LIN {X 0,Y 362.292,Z 979.123,A -85,B 0,C 180,E1 20647.364,E2 20647.364} C_VEL
LIN {X 0,Y 378.489,Z 944.913,A -85,B 0,C 180,E1 20652.896,E2 20652.896} C_VEL
LIN {X 0,Y 394.767,Z 905.956,A -85,B 0,C 180,E1 20657.324,E2 20657.324} C_VEL
LIN {X 0,Y 409.414,Z 863.634,A -85,B 0,C 180,E1 20660.691,E2 20660.691} C_VEL
LIN {X 0,Y 410.209,Z 859.007,A -85,B 0,C 180,E1 20661.092,E2 20661.092} C_VEL
LIN {X 0,Y 403.071,Z 830.26,A -85,B 0,C 180,E1 20665.806,E2 20665.806} C_VEL
LIN {X 0,Y 392.847,Z 803.519,A -85,B 0,C 180,E1 20671.168,E2 20671.168} C_VEL
LIN {X 0,Y 382.357,Z 782.646,A -85,B 0,C 180,E1 20676.647,E2 20676.647} C_VEL
LIN {X 0,Y 373.302,Z 766.723,A -85,B 0,C 180,E1 20682.27,E2 20682.27} C_VEL
LIN {X 0,Y 368.306,Z 759.241,A -85,B 0,C 180,E1 20686.159,E2 20686.159} C_VEL
LIN {X 0,Y 364.911,Z 753.277,A -85,B 0,C 180,E1 20689.83,E2 20689.83} C_VEL
LIN {X 0,Y 361.485,Z 746.529,A -85,B 0,C 180,E1 20698.795,E2 20698.795} C_VEL
LIN {X 0,Y 361.688,Z 747.798,A -85,B 0,C 180,E1 20701.421,E2 20701.421} C_VEL
LIN {X 0,Y 366.173,Z 754.902,A -85,B 0,C 180,E1 20709.074,E2 20709.074} C_VEL
LIN {X 0,Y 371.126,Z 763.095,A -85,B 0,C 180,E1 20713.499,E2 20713.499} C_VEL
LIN {X 0,Y 378.632,Z 774.835,A -85,B 0,C 180,E1 20718.367,E2 20718.367} C_VEL
LIN {X 0,Y 390.26,Z 795.362,A -85,B 0,C 180,E1 20724.362,E2 20724.362} C_VEL
LIN {X 0,Y 401.792,Z 821.282,A -85,B 0,C 180,E1 20729.832,E2 20729.832} C_VEL
LIN {X 0,Y 411.136,Z 849.862,A -85,B 0,C 180,E1 20734.599,E2 20734.599} C_VEL
LIN {X 0,Y 413.088,Z 859.947,A -85,B 0,C 180,E1 20735.992,E2 20735.992} C_VEL
LIN {X 0,Y 398.616,Z 904.569,A -85,B 0,C 180,E1 20738.996,E2 20738.996} C_VEL
LIN {X 0,Y 382.398,Z 945.744,A -85,B 0,C 180,E1 20743.057,E2 20743.057} C_VEL
LIN {X 0,Y 366.082,Z 981.986,A -85,B 0,C 180,E1 20748.161,E2 20748.161} C_VEL
LIN {X 0,Y 351.337,Z 1013.074,A -85,B 0,C 180,E1 20754.389,E2 20754.389} C_VEL
LIN {X 0,Y 339.93,Z 1037.627,A -85,B 0,C 180,E1 20761.363,E2 20761.363} C_VEL
LIN {X 0,Y 332.379,Z 1056.352,A -85,B 0,C 180,E1 20769.02,E2 20769.02} C_VEL
LIN {X 0,Y 328.863,Z 1068.693,A -85,B 0,C 180,E1 20776.678,E2 20776.678} C_VEL
LIN {X 0,Y 328.034,Z 1074.064,A -85,B 0,C 180,E1 20782.033,E2 20782.033} C_VEL
LIN {X 0,Y 328.003,Z 1077.219,A -85,B 0,C 180,E1 20789.999,E2 20789.999} C_VEL
LIN {X 0,Y 327.96,Z 1074.585,A -85,B 0,C 180,E1 20797.967,E2 20797.967} C_VEL
LIN {X 0,Y 329.425,Z 1067.671,A -85,B 0,C 180,E1 20804.999,E2 20804.999} C_VEL
LIN {X 0,Y 334.439,Z 1053.272,A -85,B 0,C 180,E1 20813.357,E2 20813.357} C_VEL
LIN {X 0,Y 344.133,Z 1032.137,A -85,B 0,C 180,E1 20821.314,E2 20821.314} C_VEL
LIN {X 0,Y 357.491,Z 1005.639,A -85,B 0,C 180,E1 20828.176,E2 20828.176} C_VEL
LIN {X 0,Y 372.702,Z 975.355,A -85,B 0,C 180,E1 20833.725,E2 20833.725} C_VEL
LIN {X 0,Y 388.88,Z 940.762,A -85,B 0,C 180,E1 20838.265,E2 20838.265} C_VEL
LIN {X 0,Y 404.573,Z 902.35,A -85,B 0,C 180,E1 20841.866,E2 20841.866} C_VEL
LIN {X 0,Y 418.082,Z 861.927,A -85,B 0,C 180,E1 20844.559,E2 20844.559} C_VEL
LIN {X 0,Y 409.957,Z 833.961,A -85,B 0,C 180,E1 20849.35,E2 20849.35} C_VEL
LIN {X 0,Y 399.624,Z 808.583,A -85,B 0,C 180,E1 20854.842,E2 20854.842} C_VEL
LIN {X 0,Y 393.435,Z 796.515,A -85,B 0,C 180,E1 20858.246,E2 20858.246} C_VEL
LIN {X 0,Y 389.709,Z 795.233,A -85,B 0,C 180,E1 20859.866,E2 20859.866} C_VEL
LIN {X 0,Y 386.052,Z 794.568,A -85,B 0,C 180,E1 20861.545,E2 20861.545} C_VEL
LIN {X 0,Y 378.893,Z 781.987,A -85,B 0,C 180,E1 20867.338,E2 20867.338} C_VEL
LIN {X 0,Y 375.953,Z 776.169,A -85,B 0,C 180,E1 20871.018,E2 20871.018} C_VEL
LIN {X 0,Y 373.294,Z 769.834,A -85,B 0,C 180,E1 20879.423,E2 20879.423} C_VEL
LIN {X 0,Y 376.486,Z 777.904,A -85,B 0,C 180,E1 20888.613,E2 20888.613} C_VEL
LIN {X 0,Y 380.579,Z 785.858,A -85,B 0,C 180,E1 20893.093,E2 20893.093} C_VEL
LIN {X 0,Y 386.293,Z 796.722,A -85,B 0,C 180,E1 20897.704,E2 20897.704} C_VEL
LIN {X 0,Y 394.613,Z 814.838,A -85,B 0,C 180,E1 20903.244,E2 20903.244} C_VEL
LIN {X 0,Y 402.714,Z 837.776,A -85,B 0,C 180,E1 20908.5,E2 20908.5} C_VEL
LIN {X 0,Y 408.935,Z 862.896,A -85,B 0,C 180,E1 20913.197,E2 20913.197} C_VEL
LIN {X 0,Y 408.939,Z 868.346,A -85,B 0,C 180,E1 20913.956,E2 20913.956} C_VEL
LIN {X 0,Y 394.051,Z 907.639,A -85,B 0,C 180,E1 20917.064,E2 20917.064} C_VEL
LIN {X 0,Y 376.826,Z 945.755,A -85,B 0,C 180,E1 20921.379,E2 20921.379} C_VEL
LIN {X 0,Y 359.627,Z 979.236,A -85,B 0,C 180,E1 20926.786,E2 20926.786} C_VEL
LIN {X 0,Y 343.841,Z 1008.047,A -85,B 0,C 180,E1 20933.49,E2 20933.49} C_VEL
LIN {X 0,Y 332.266,Z 1029.329,A -85,B 0,C 180,E1 20940.642,E2 20940.642} C_VEL
LIN {X 0,Y 325.06,Z 1044.409,A -85,B 0,C 180,E1 20948.104,E2 20948.104} C_VEL
LIN {X 0,Y 321.603,Z 1053.264,A -85,B 0,C 180,E1 20954.699,E2 20954.699} C_VEL
LIN {X 0,Y 319.956,Z 1058.652,A -85,B 0,C 180,E1 20961.833,E2 20961.833} C_VEL
LIN {X 0,Y 320.103,Z 1059.662,A -85,B 0,C 180,E1 20970.001,E2 20970.001} C_VEL
LIN {X 0,Y 320.678,Z 1055.234,A -85,B 0,C 180,E1 20978.151,E2 20978.151} C_VEL
LIN {X 0,Y 323.464,Z 1046.348,A -85,B 0,C 180,E1 20985.629,E2 20985.629} C_VEL
LIN {X 0,Y 329.929,Z 1030.99,A -85,B 0,C 180,E1 20993.549,E2 20993.549} C_VEL
LIN {X 0,Y 340.701,Z 1009.055,A -85,B 0,C 180,E1 21001.137,E2 21001.137} C_VEL
LIN {X 0,Y 354.739,Z 981.771,A -85,B 0,C 180,E1 21007.676,E2 21007.676} C_VEL
LIN {X 0,Y 370.156,Z 950.547,A -85,B 0,C 180,E1 21012.981,E2 21012.981} C_VEL
LIN {X 0,Y 385.613,Z 915.656,A -85,B 0,C 180,E1 21017.257,E2 21017.257} C_VEL
LIN {X 0,Y 400.393,Z 876.252,A -85,B 0,C 180,E1 21020.729,E2 21020.729} C_VEL
LIN {X 0,Y 404.623,Z 862.747,A -85,B 0,C 180,E1 21021.704,E2 21021.704} C_VEL
LIN {X 0,Y 397.926,Z 834.187,A -85,B 0,C 180,E1 21026.549,E2 21026.549} C_VEL
LIN {X 0,Y 388.172,Z 807.746,A -85,B 0,C 180,E1 21032.061,E2 21032.061} C_VEL
LIN {X 0,Y 377.812,Z 785.992,A -85,B 0,C 180,E1 21038.078,E2 21038.078} C_VEL
LIN {X 0,Y 369.588,Z 772.075,A -85,B 0,C 180,E1 21043.714,E2 21043.714} C_VEL
LIN {X 0,Y 366.487,Z 766.793,A -85,B 0,C 180,E1 21046.394,E2 21046.394} C_VEL
LIN {X 0,Y 363.309,Z 760.907,A -85,B 0,C 180,E1 21050.088,E2 21050.088} C_VEL
LIN {X 0,Y 360.349,Z 754.316,A -85,B 0,C 180,E1 21058.791,E2 21058.791} C_VEL
LIN {X 0,Y 360.53,Z 755.742,A -85,B 0,C 180,E1 21061.426,E2 21061.426} C_VEL
LIN {X 0,Y 364.652,Z 762.65,A -85,B 0,C 180,E1 21068.886,E2 21068.886} C_VEL
LIN {X 0,Y 369.221,Z 770.705,A -85,B 0,C 180,E1 21073.268,E2 21073.268} C_VEL
LIN {X 0,Y 376.265,Z 782.283,A -85,B 0,C 180,E1 21078.107,E2 21078.107} C_VEL
LIN {X 0,Y 386.877,Z 802.016,A -85,B 0,C 180,E1 21083.973,E2 21083.973} C_VEL
LIN {X 0,Y 397.578,Z 827.186,A -85,B 0,C 180,E1 21089.384,E2 21089.384} C_VEL
LIN {X 0,Y 405.873,Z 854.347,A -85,B 0,C 180,E1 21094.054,E2 21094.054} C_VEL
LIN {X 0,Y 407.499,Z 862.634,A -85,B 0,C 180,E1 21095.268,E2 21095.268} C_VEL
LIN {X 0,Y 393.211,Z 905.194,A -85,B 0,C 180,E1 21098.169,E2 21098.169} C_VEL
LIN {X 0,Y 376.403,Z 946.465,A -85,B 0,C 180,E1 21102.286,E2 21102.286} C_VEL
LIN {X 0,Y 359.289,Z 983.156,A -85,B 0,C 180,E1 21107.557,E2 21107.557} C_VEL
LIN {X 0,Y 344.063,Z 1014.027,A -85,B 0,C 180,E1 21113.906,E2 21113.906} C_VEL
LIN {X 0,Y 331.885,Z 1039.267,A -85,B 0,C 180,E1 21121.35,E2 21121.35} C_VEL
LIN {X 0,Y 324.4,Z 1057.268,A -85,B 0,C 180,E1 21129.096,E2 21129.096} C_VEL
LIN {X 0,Y 321.064,Z 1068.453,A -85,B 0,C 180,E1 21136.348,E2 21136.348} C_VEL
LIN {X 0,Y 319.869,Z 1075.333,A -85,B 0,C 180,E1 21144.149,E2 21144.149} C_VEL
LIN {X 0,Y 320.101,Z 1077.005,A -85,B 0,C 180,E1 21149.999,E2 21149.999} C_VEL
LIN {X 0,Y 320.082,Z 1074.387,A -85,B 0,C 180,E1 21158.164,E2 21158.164} C_VEL
LIN {X 0,Y 321.634,Z 1067.481,A -85,B 0,C 180,E1 21165.371,E2 21165.371} C_VEL
LIN {X 0,Y 326.987,Z 1053.1,A -85,B 0,C 180,E1 21173.922,E2 21173.922} C_VEL
LIN {X 0,Y 336.463,Z 1033.335,A -85,B 0,C 180,E1 21181.593,E2 21181.593} C_VEL
LIN {X 0,Y 349.526,Z 1008.452,A -85,B 0,C 180,E1 21188.334,E2 21188.334} C_VEL
LIN {X 0,Y 365.019,Z 978.964,A -85,B 0,C 180,E1 21194.014,E2 21194.014} C_VEL
LIN {X 0,Y 382.343,Z 943.482,A -85,B 0,C 180,E1 21198.854,E2 21198.854} C_VEL
LIN {X 0,Y 399.125,Z 903.877,A -85,B 0,C 180,E1 21202.651,E2 21202.651} C_VEL
LIN {X 0,Y 412.314,Z 865.921,A -85,B 0,C 180,E1 21205.219,E2 21205.219} C_VEL
LIN {X 0,Y 406.165,Z 841.459,A -85,B 0,C 180,E1 21209.45,E2 21209.45} C_VEL
LIN {X 0,Y 397.177,Z 817.77,A -85,B 0,C 180,E1 21214.586,E2 21214.586} C_VEL
LIN {X 0,Y 387.984,Z 798.501,A -85,B 0,C 180,E1 21220.169,E2 21220.169} C_VEL
LIN {X 0,Y 386.052,Z 794.568,A -85,B 0,C 180,E1 21221.545,E2 21221.545} C_VEL
LIN {X 0,Y 381.552,Z 792.796,A -85,B 0,C 180,E1 21224.065,E2 21224.065} C_VEL
LIN {X 0,Y 377.763,Z 790.787,A -85,B 0,C 180,E1 21226.627,E2 21226.627} C_VEL
LIN {X 0,Y 373.896,Z 783.707,A -85,B 0,C 180,E1 21231.262,E2 21231.262} C_VEL
LIN {X 0,Y 371.646,Z 777.561,A -85,B 0,C 180,E1 21239.42,E2 21239.42} C_VEL
LIN {X 0,Y 374.445,Z 785.549,A -85,B 0,C 180,E1 21248.44,E2 21248.44} C_VEL
LIN {X 0,Y 378.451,Z 793.827,A -85,B 0,C 180,E1 21253.168,E2 21253.168} C_VEL
LIN {X 0,Y 385.176,Z 807.455,A -85,B 0,C 180,E1 21258.733,E2 21258.733} C_VEL
LIN {X 0,Y 393.599,Z 828.768,A -85,B 0,C 180,E1 21264.757,E2 21264.757} C_VEL
LIN {X 0,Y 400.924,Z 854.087,A -85,B 0,C 180,E1 21270.215,E2 21270.215} C_VEL
LIN {X 0,Y 403.718,Z 870.502,A -85,B 0,C 180,E1 21273.16,E2 21273.16} C_VEL
LIN {X 0,Y 388.089,Z 910.178,A -85,B 0,C 180,E1 21276.357,E2 21276.357} C_VEL
LIN {X 0,Y 371.333,Z 946.125,A -85,B 0,C 180,E1 21280.481,E2 21280.481} C_VEL
LIN {X 0,Y 353.721,Z 979.362,A -85,B 0,C 180,E1 21285.889,E2 21285.889} C_VEL
LIN {X 0,Y 337.231,Z 1008.176,A -85,B 0,C 180,E1 21292.654,E2 21292.654} C_VEL
LIN {X 0,Y 324.304,Z 1031.094,A -85,B 0,C 180,E1 21300.619,E2 21300.619} C_VEL
LIN {X 0,Y 316.807,Z 1046.279,A -85,B 0,C 180,E1 21308.614,E2 21308.614} C_VEL
LIN {X 0,Y 313.255,Z 1055.058,A -85,B 0,C 180,E1 21316.004,E2 21316.004} C_VEL
LIN {X 0,Y 311.855,Z 1059.838,A -85,B 0,C 180,E1 21324.424,E2 21324.424} C_VEL
LIN {X 0,Y 312.202,Z 1059.876,A -85,B 0,C 180,E1 21330.001,E2 21330.001} C_VEL
LIN {X 0,Y 312.815,Z 1055.471,A -85,B 0,C 180,E1 21338.358,E2 21338.358} C_VEL
LIN {X 0,Y 316.05,Z 1045.9,A -85,B 0,C 180,E1 21346.456,E2 21346.456} C_VEL
LIN {X 0,Y 323.52,Z 1029.351,A -85,B 0,C 180,E1 21354.935,E2 21354.935} C_VEL
LIN {X 0,Y 335.046,Z 1007.205,A -85,B 0,C 180,E1 21362.488,E2 21362.488} C_VEL
LIN {X 0,Y 350.26,Z 978.777,A -85,B 0,C 180,E1 21369.162,E2 21369.162} C_VEL
LIN {X 0,Y 367.716,Z 944.063,A -85,B 0,C 180,E1 21374.814,E2 21374.814} C_VEL
LIN {X 0,Y 384.851,Z 905.214,A -85,B 0,C 180,E1 21379.213,E2 21379.213} C_VEL
LIN {X 0,Y 398.911,Z 865.969,A -85,B 0,C 180,E1 21382.393,E2 21382.393} C_VEL
LIN {X 0,Y 392.738,Z 838.129,A -85,B 0,C 180,E1 21387.299,E2 21387.299} C_VEL
LIN {X 0,Y 384.055,Z 813.16,A -85,B 0,C 180,E1 21392.693,E2 21392.693} C_VEL
LIN {X 0,Y 374.542,Z 792.411,A -85,B 0,C 180,E1 21398.641,E2 21398.641} C_VEL
LIN {X 0,Y 367.203,Z 779.273,A -85,B 0,C 180,E1 21404.071,E2 21404.071} C_VEL
LIN {X 0,Y 364.404,Z 774.124,A -85,B 0,C 180,E1 21406.795,E2 21406.795} C_VEL
LIN {X 0,Y 361.587,Z 768.514,A -85,B 0,C 180,E1 21410.345,E2 21410.345} C_VEL
LIN {X 0,Y 359.009,Z 762.081,A -85,B 0,C 180,E1 21418.786,E2 21418.786} C_VEL
LIN {X 0,Y 359.112,Z 763.793,A -85,B 0,C 180,E1 21421.507,E2 21421.507} C_VEL
LIN {X 0,Y 362.933,Z 770.376,A -85,B 0,C 180,E1 21428.701,E2 21428.701} C_VEL
LIN {X 0,Y 367.348,Z 778.375,A -85,B 0,C 180,E1 21433.109,E2 21433.109} C_VEL
LIN {X 0,Y 374.694,Z 791.276,A -85,B 0,C 180,E1 21438.414,E2 21438.414} C_VEL
LIN {X 0,Y 384.323,Z 810.555,A -85,B 0,C 180,E1 21444.027,E2 21444.027} C_VEL
LIN {X 0,Y 393.949,Z 835.151,A -85,B 0,C 180,E1 21449.365,E2 21449.365} C_VEL
LIN {X 0,Y 401.658,Z 863.672,A -85,B 0,C 180,E1 21454.271,E2 21454.271} C_VEL
LIN {X 0,Y 400.678,Z 869.274,A -85,B 0,C 180,E1 21454.754,E2 21454.754} C_VEL
LIN {X 0,Y 386.515,Z 909.286,A -85,B 0,C 180,E1 21457.629,E2 21457.629} C_VEL
LIN {X 0,Y 370.756,Z 946.599,A -85,B 0,C 180,E1 21461.421,E2 21461.421} C_VEL
LIN {X 0,Y 353.334,Z 982.829,A -85,B 0,C 180,E1 21466.667,E2 21466.667} C_VEL
LIN {X 0,Y 337.487,Z 1013.726,A -85,B 0,C 180,E1 21473.088,E2 21473.088} C_VEL
LIN {X 0,Y 324.761,Z 1038.991,A -85,B 0,C 180,E1 21480.661,E2 21480.661} C_VEL
LIN {X 0,Y 316.799,Z 1057.006,A -85,B 0,C 180,E1 21488.57,E2 21488.57} C_VEL
LIN {X 0,Y 313.263,Z 1068.213,A -85,B 0,C 180,E1 21496.002,E2 21496.002} C_VEL
LIN {X 0,Y 312.271,Z 1073.611,A -85,B 0,C 180,E1 21501.628,E2 21501.628} C_VEL
LIN {X 0,Y 312.2,Z 1076.792,A -85,B 0,C 180,E1 21509.999,E2 21509.999} C_VEL
LIN {X 0,Y 312,Z 1075.68,A -85,B 0,C 180,E1 21515.573,E2 21515.573} C_VEL
LIN {X 0,Y 312.86,Z 1070.82,A -85,B 0,C 180,E1 21522.588,E2 21522.588} C_VEL
LIN {X 0,Y 316.908,Z 1058.955,A -85,B 0,C 180,E1 21531.328,E2 21531.328} C_VEL
LIN {X 0,Y 324.965,Z 1041.713,A -85,B 0,C 180,E1 21539.316,E2 21539.316} C_VEL
LIN {X 0,Y 337.275,Z 1018.994,A -85,B 0,C 180,E1 21546.535,E2 21546.535} C_VEL
LIN {X 0,Y 353.149,Z 990.205,A -85,B 0,C 180,E1 21552.937,E2 21552.937} C_VEL
LIN {X 0,Y 370.92,Z 956.236,A -85,B 0,C 180,E1 21558.21,E2 21558.21} C_VEL
LIN {X 0,Y 388.772,Z 917.347,A -85,B 0,C 180,E1 21562.434,E2 21562.434} C_VEL
LIN {X 0,Y 405.167,Z 874.138,A -85,B 0,C 180,E1 21565.668,E2 21565.668} C_VEL
LIN {X 0,Y 406.897,Z 868.272,A -85,B 0,C 180,E1 21566.043,E2 21566.043} C_VEL
LIN {X 0,Y 399.682,Z 840.893,A -85,B 0,C 180,E1 21571.154,E2 21571.154} C_VEL
LIN {X 0,Y 390.951,Z 818.002,A -85,B 0,C 180,E1 21576.595,E2 21576.595} C_VEL
LIN {X 0,Y 382.734,Z 800.851,A -85,B 0,C 180,E1 21582.213,E2 21582.213} C_VEL
LIN {X 0,Y 377.763,Z 790.787,A -85,B 0,C 180,E1 21586.627,E2 21586.627} C_VEL
LIN {X 0,Y 375.444,Z 789.408,A -85,B 0,C 180,E1 21588.567,E2 21588.567} C_VEL
LIN {X 0,Y 371.55,Z 790.969,A -85,B 0,C 180,E1 21591.926,E2 21591.926} C_VEL
LIN {X 0,Y 369.81,Z 785.22,A -85,B 0,C 180,E1 21599.417,E2 21599.417} C_VEL
LIN {X 0,Y 372.248,Z 793.063,A -85,B 0,C 180,E1 21608.269,E2 21608.269} C_VEL
LIN {X 0,Y 376.132,Z 801.593,A -85,B 0,C 180,E1 21613.158,E2 21613.158} C_VEL
LIN {X 0,Y 382.063,Z 814.674,A -85,B 0,C 180,E1 21618.504,E2 21618.504} C_VEL
LIN {X 0,Y 389.671,Z 835.188,A -85,B 0,C 180,E1 21624.41,E2 21624.41} C_VEL
LIN {X 0,Y 396.096,Z 859.74,A -85,B 0,C 180,E1 21629.83,E2 21629.83} C_VEL
LIN {X 0,Y 397.996,Z 874.273,A -85,B 0,C 180,E1 21632.452,E2 21632.452} C_VEL
LIN {X 0,Y 381.674,Z 913.982,A -85,B 0,C 180,E1 21635.764,E2 21635.764} C_VEL
LIN {X 0,Y 364.607,Z 949.038,A -85,B 0,C 180,E1 21639.922,E2 21639.922} C_VEL
LIN {X 0,Y 346.941,Z 981.077,A -85,B 0,C 180,E1 21645.286,E2 21645.286} C_VEL
LIN {X 0,Y 330.626,Z 1008.494,A -85,B 0,C 180,E1 21651.849,E2 21651.849} C_VEL
LIN {X 0,Y 317.712,Z 1030.406,A -85,B 0,C 180,E1 21659.519,E2 21659.519} C_VEL
LIN {X 0,Y 309.271,Z 1046.4,A -85,B 0,C 180,E1 21668.035,E2 21668.035} C_VEL
LIN {X 0,Y 305.48,Z 1055.247,A -85,B 0,C 180,E1 21675.64,E2 21675.64} C_VEL
LIN {X 0,Y 303.978,Z 1060.043,A -85,B 0,C 180,E1 21684.279,E2 21684.279} C_VEL
LIN {X 0,Y 304.298,Z 1060.09,A -85,B 0,C 180,E1 21690.001,E2 21690.001} C_VEL
LIN {X 0,Y 304.973,Z 1055.708,A -85,B 0,C 180,E1 21698.574,E2 21698.574} C_VEL
LIN {X 0,Y 308.204,Z 1046.67,A -85,B 0,C 180,E1 21706.554,E2 21706.554} C_VEL
LIN {X 0,Y 315.541,Z 1031.045,A -85,B 0,C 180,E1 21714.946,E2 21714.946} C_VEL
LIN {X 0,Y 327.661,Z 1008.596,A -85,B 0,C 180,E1 21722.919,E2 21722.919} C_VEL
LIN {X 0,Y 343.258,Z 980.565,A -85,B 0,C 180,E1 21729.704,E2 21729.704} C_VEL
LIN {X 0,Y 360.311,Z 947.915,A -85,B 0,C 180,E1 21735.214,E2 21735.214} C_VEL
LIN {X 0,Y 376.602,Z 912.738,A -85,B 0,C 180,E1 21739.422,E2 21739.422} C_VEL
LIN {X 0,Y 391.363,Z 874.905,A -85,B 0,C 180,E1 21742.687,E2 21742.687} C_VEL
LIN {X 0,Y 393.177,Z 868.813,A -85,B 0,C 180,E1 21743.17,E2 21743.17} C_VEL
LIN {X 0,Y 387.824,Z 842.891,A -85,B 0,C 180,E1 21747.91,E2 21747.91} C_VEL
LIN {X 0,Y 379.913,Z 818.578,A -85,B 0,C 180,E1 21753.358,E2 21753.358} C_VEL
LIN {X 0,Y 371.017,Z 798.402,A -85,B 0,C 180,E1 21759.377,E2 21759.377} C_VEL
LIN {X 0,Y 364.246,Z 785.132,A -85,B 0,C 180,E1 21765.016,E2 21765.016} C_VEL
LIN {X 0,Y 359.792,Z 776.133,A -85,B 0,C 180,E1 21770.517,E2 21770.517} C_VEL
LIN {X 0,Y 357.517,Z 769.834,A -85,B 0,C 180,E1 21778.781,E2 21778.781} C_VEL
LIN {X 0,Y 357.6,Z 771.651,A -85,B 0,C 180,E1 21781.513,E2 21781.513} C_VEL
LIN {X 0,Y 361.081,Z 777.893,A -85,B 0,C 180,E1 21788.442,E2 21788.442} C_VEL
LIN {X 0,Y 365.542,Z 786.619,A -85,B 0,C 180,E1 21793.252,E2 21793.252} C_VEL
LIN {X 0,Y 373.085,Z 800.596,A -85,B 0,C 180,E1 21798.881,E2 21798.881} C_VEL
LIN {X 0,Y 382.115,Z 820.42,A -85,B 0,C 180,E1 21804.478,E2 21804.478} C_VEL
LIN {X 0,Y 391.113,Z 846.136,A -85,B 0,C 180,E1 21809.919,E2 21809.919} C_VEL
LIN {X 0,Y 396.181,Z 868.798,A -85,B 0,C 180,E1 21813.805,E2 21813.805} C_VEL
LIN {X 0,Y 381.692,Z 908.704,A -85,B 0,C 180,E1 21816.651,E2 21816.651} C_VEL
LIN {X 0,Y 365.156,Z 946.86,A -85,B 0,C 180,E1 21820.548,E2 21820.548} C_VEL
LIN {X 0,Y 347.469,Z 982.502,A -85,B 0,C 180,E1 21825.748,E2 21825.748} C_VEL
LIN {X 0,Y 330.953,Z 1013.423,A -85,B 0,C 180,E1 21832.233,E2 21832.233} C_VEL
LIN {X 0,Y 317.66,Z 1038.753,A -85,B 0,C 180,E1 21839.956,E2 21839.956} C_VEL
LIN {X 0,Y 309.24,Z 1056.745,A -85,B 0,C 180,E1 21848.021,E2 21848.021} C_VEL
LIN {X 0,Y 305.486,Z 1067.973,A -85,B 0,C 180,E1 21855.638,E2 21855.638} C_VEL
LIN {X 0,Y 304.378,Z 1073.384,A -85,B 0,C 180,E1 21861.409,E2 21861.409} C_VEL
LIN {X 0,Y 304.084,Z 1076.176,A -85,B 0,C 180,E1 21867.142,E2 21867.142} C_VEL
LIN {X 0,Y 304.154,Z 1076.34,A -85,B 0,C 180,E1 21872.855,E2 21872.855} C_VEL
LIN {X 0,Y 304.681,Z 1071.869,A -85,B 0,C 180,E1 21881.474,E2 21881.474} C_VEL
LIN {X 0,Y 307.706,Z 1062.746,A -85,B 0,C 180,E1 21889.415,E2 21889.415} C_VEL
LIN {X 0,Y 315.062,Z 1046.87,A -85,B 0,C 180,E1 21897.862,E2 21897.862} C_VEL
LIN {X 0,Y 327.148,Z 1024.968,A -85,B 0,C 180,E1 21905.659,E2 21905.659} C_VEL
LIN {X 0,Y 342.155,Z 999.138,A -85,B 0,C 180,E1 21912.049,E2 21912.049} C_VEL
LIN {X 0,Y 359.688,Z 967.325,A -85,B 0,C 180,E1 21917.623,E2 21917.623} C_VEL
LIN {X 0,Y 377.978,Z 930.551,A -85,B 0,C 180,E1 21922.12,E2 21922.12} C_VEL
LIN {X 0,Y 395.625,Z 888.368,A -85,B 0,C 180,E1 21925.681,E2 21925.681} C_VEL
LIN {X 0,Y 401.289,Z 870.961,A -85,B 0,C 180,E1 21926.907,E2 21926.907} C_VEL
LIN {X 0,Y 394.704,Z 844.822,A -85,B 0,C 180,E1 21932.01,E2 21932.01} C_VEL
LIN {X 0,Y 387.452,Z 824.55,A -85,B 0,C 180,E1 21936.981,E2 21936.981} C_VEL
LIN {X 0,Y 379.732,Z 807.552,A -85,B 0,C 180,E1 21942.696,E2 21942.696} C_VEL
LIN {X 0,Y 374.133,Z 796.472,A -85,B 0,C 180,E1 21948.091,E2 21948.091} C_VEL
LIN {X 0,Y 371.851,Z 791.226,A -85,B 0,C 180,E1 21951.509,E2 21951.509} C_VEL
LIN {X 0,Y 371.55,Z 790.969,A -85,B 0,C 180,E1 21951.926,E2 21951.926} C_VEL
LIN {X 0,Y 367.716,Z 794.575,A -85,B 0,C 180,E1 21956.96,E2 21956.96} C_VEL
LIN {X 0,Y 367.692,Z 794.354,A -85,B 0,C 180,E1 21957.299,E2 21957.299} C_VEL
LIN {X 0,Y 367.809,Z 793.085,A -85,B 0,C 180,E1 21959.709,E2 21959.709} C_VEL
LIN {X 0,Y 369.902,Z 800.655,A -85,B 0,C 180,E1 21968.137,E2 21968.137} C_VEL
LIN {X 0,Y 373.811,Z 809.63,A -85,B 0,C 180,E1 21973.364,E2 21973.364} C_VEL
LIN {X 0,Y 379.892,Z 824.601,A -85,B 0,C 180,E1 21979.218,E2 21979.218} C_VEL
LIN {X 0,Y 386.19,Z 843.965,A -85,B 0,C 180,E1 21984.664,E2 21984.664} C_VEL
LIN {X 0,Y 391.612,Z 867.493,A -85,B 0,C 180,E1 21989.886,E2 21989.886} C_VEL
LIN {X 0,Y 392.542,Z 877.55,A -85,B 0,C 180,E1 21991.695,E2 21991.695} C_VEL
LIN {X 0,Y 374.635,Z 919.26,A -85,B 0,C 180,E1 21995.299,E2 21995.299} C_VEL
LIN {X 0,Y 355.715,Z 956.036,A -85,B 0,C 180,E1 21999.932,E2 21999.932} C_VEL
LIN {X 0,Y 336.753,Z 988.514,A -85,B 0,C 180,E1 22005.858,E2 22005.858} C_VEL
LIN {X 0,Y 319.679,Z 1016.056,A -85,B 0,C 180,E1 22013.275,E2 22013.275} C_VEL
LIN {X 0,Y 307.364,Z 1036.102,A -85,B 0,C 180,E1 22021.351,E2 22021.351} C_VEL
LIN {X 0,Y 300.492,Z 1049.088,A -85,B 0,C 180,E1 22029.33,E2 22029.33} C_VEL
LIN {X 0,Y 297.28,Z 1056.632,A -85,B 0,C 180,E1 22036.758,E2 22036.758} C_VEL
LIN {X 0,Y 296.077,Z 1060.249,A -85,B 0,C 180,E1 22044.126,E2 22044.126} C_VEL
LIN {X 0,Y 296.423,Z 1060.304,A -85,B 0,C 180,E1 22050.001,E2 22050.001} C_VEL
LIN {X 0,Y 297.119,Z 1055.945,A -85,B 0,C 180,E1 22058.803,E2 22058.803} C_VEL
LIN {X 0,Y 300.234,Z 1047.675,A -85,B 0,C 180,E1 22066.446,E2 22066.446} C_VEL
LIN {X 0,Y 308.147,Z 1031.513,A -85,B 0,C 180,E1 22075.488,E2 22075.488} C_VEL
LIN {X 0,Y 320.281,Z 1009.967,A -85,B 0,C 180,E1 22083.371,E2 22083.371} C_VEL
LIN {X 0,Y 335.637,Z 983.43,A -85,B 0,C 180,E1 22090.045,E2 22090.045} C_VEL
LIN {X 0,Y 352.749,Z 952.071,A -85,B 0,C 180,E1 22095.58,E2 22095.58} C_VEL
LIN {X 0,Y 369.853,Z 916.901,A -85,B 0,C 180,E1 22099.969,E2 22099.969} C_VEL
LIN {X 0,Y 386.263,Z 876.398,A -85,B 0,C 180,E1 22103.549,E2 22103.549} C_VEL
LIN {X 0,Y 387.438,Z 871.073,A -85,B 0,C 180,E1 22104.072,E2 22104.072} C_VEL
LIN {X 0,Y 382.374,Z 845.472,A -85,B 0,C 180,E1 22108.984,E2 22108.984} C_VEL
LIN {X 0,Y 374.843,Z 821.652,A -85,B 0,C 180,E1 22114.621,E2 22114.621} C_VEL
LIN {X 0,Y 366.236,Z 801.259,A -85,B 0,C 180,E1 22121.227,E2 22121.227} C_VEL
LIN {X 0,Y 360.139,Z 789.002,A -85,B 0,C 180,E1 22127.266,E2 22127.266} C_VEL
LIN {X 0,Y 357.651,Z 783.59,A -85,B 0,C 180,E1 22130.904,E2 22130.904} C_VEL
LIN {X 0,Y 355.871,Z 777.565,A -85,B 0,C 180,E1 22138.776,E2 22138.776} C_VEL
LIN {X 0,Y 355.867,Z 779.474,A -85,B 0,C 180,E1 22141.521,E2 22141.521} C_VEL
LIN {X 0,Y 359.031,Z 785.522,A -85,B 0,C 180,E1 22148.262,E2 22148.262} C_VEL
LIN {X 0,Y 364.796,Z 796.586,A -85,B 0,C 180,E1 22154.351,E2 22154.351} C_VEL
LIN {X 0,Y 372.674,Z 813.272,A -85,B 0,C 180,E1 22160.34,E2 22160.34} C_VEL
LIN {X 0,Y 381.171,Z 834.656,A -85,B 0,C 180,E1 22165.928,E2 22165.928} C_VEL
LIN {X 0,Y 388.523,Z 860.399,A -85,B 0,C 180,E1 22171.069,E2 22171.069} C_VEL
LIN {X 0,Y 390.453,Z 872.327,A -85,B 0,C 180,E1 22173.064,E2 22173.064} C_VEL
LIN {X 0,Y 375,Z 912.962,A -85,B 0,C 180,E1 22176.077,E2 22176.077} C_VEL
LIN {X 0,Y 358.004,Z 950.253,A -85,B 0,C 180,E1 22180.031,E2 22180.031} C_VEL
LIN {X 0,Y 340.843,Z 983.627,A -85,B 0,C 180,E1 22185.057,E2 22185.057} C_VEL
LIN {X 0,Y 324.562,Z 1013.124,A -85,B 0,C 180,E1 22191.354,E2 22191.354} C_VEL
LIN {X 0,Y 310.472,Z 1038.723,A -85,B 0,C 180,E1 22199.3,E2 22199.3} C_VEL
LIN {X 0,Y 301.093,Z 1057.981,A -85,B 0,C 180,E1 22208.297,E2 22208.297} C_VEL
LIN {X 0,Y 297.265,Z 1069.338,A -85,B 0,C 180,E1 22216.737,E2 22216.737} C_VEL
LIN {X 0,Y 296.205,Z 1074.897,A -85,B 0,C 180,E1 22224.126,E2 22224.126} C_VEL
LIN {X 0,Y 296.423,Z 1076.365,A -85,B 0,C 180,E1 22229.999,E2 22229.999} C_VEL
LIN {X 0,Y 296.203,Z 1075.273,A -85,B 0,C 180,E1 22235.872,E2 22235.872} C_VEL
LIN {X 0,Y 297.249,Z 1070.433,A -85,B 0,C 180,E1 22243.261,E2 22243.261} C_VEL
LIN {X 0,Y 301.346,Z 1059.603,A -85,B 0,C 180,E1 22251.82,E2 22251.82} C_VEL
LIN {X 0,Y 309.853,Z 1043.166,A -85,B 0,C 180,E1 22260.081,E2 22260.081} C_VEL
LIN {X 0,Y 323.6,Z 1019.938,A -85,B 0,C 180,E1 22267.924,E2 22267.924} C_VEL
LIN {X 0,Y 341.173,Z 990.427,A -85,B 0,C 180,E1 22274.717,E2 22274.717} C_VEL
LIN {X 0,Y 360.349,Z 956.096,A -85,B 0,C 180,E1 22280.126,E2 22280.126} C_VEL
LIN {X 0,Y 378.763,Z 918.326,A -85,B 0,C 180,E1 22284.264,E2 22284.264} C_VEL
LIN {X 0,Y 395.934,Z 874.763,A -85,B 0,C 180,E1 22287.604,E2 22287.604} C_VEL
LIN {X 0,Y 390.025,Z 849.8,A -85,B 0,C 180,E1 22292.629,E2 22292.629} C_VEL
LIN {X 0,Y 383.023,Z 829.214,A -85,B 0,C 180,E1 22297.927,E2 22297.927} C_VEL
LIN {X 0,Y 376.704,Z 814.491,A -85,B 0,C 180,E1 22303.048,E2 22303.048} C_VEL
LIN {X 0,Y 371.567,Z 803.589,A -85,B 0,C 180,E1 22308.462,E2 22308.462} C_VEL
LIN {X 0,Y 369.331,Z 798.513,A -85,B 0,C 180,E1 22312.011,E2 22312.011} C_VEL
LIN {X 0,Y 367.692,Z 794.354,A -85,B 0,C 180,E1 22317.299,E2 22317.299} C_VEL
LIN {X 0,Y 366.906,Z 796.204,A -85,B 0,C 180,E1 22319.31,E2 22319.31} C_VEL
LIN {X 0,Y 365.413,Z 803.386,A -85,B 0,C 180,E1 22322.634,E2 22322.634} C_VEL
LIN {X 0,Y 367.354,Z 807.642,A -85,B 0,C 180,E1 22327.723,E2 22327.723} C_VEL
LIN {X 0,Y 371.853,Z 819.017,A -85,B 0,C 180,E1 22334.157,E2 22334.157} C_VEL
LIN {X 0,Y 377.496,Z 834.673,A -85,B 0,C 180,E1 22339.955,E2 22339.955} C_VEL
LIN {X 0,Y 383.099,Z 854.934,A -85,B 0,C 180,E1 22345.483,E2 22345.483} C_VEL
LIN {X 0,Y 387.383,Z 879.467,A -85,B 0,C 180,E1 22350.774,E2 22350.774} C_VEL
LIN {X 0,Y 369.335,Z 920.681,A -85,B 0,C 180,E1 22354.424,E2 22354.424} C_VEL
LIN {X 0,Y 349.51,Z 957.953,A -85,B 0,C 180,E1 22359.195,E2 22359.195} C_VEL
LIN {X 0,Y 329.765,Z 990.471,A -85,B 0,C 180,E1 22365.289,E2 22365.289} C_VEL
LIN {X 0,Y 312.439,Z 1017.251,A -85,B 0,C 180,E1 22372.747,E2 22372.747} C_VEL
LIN {X 0,Y 299.45,Z 1037.569,A -85,B 0,C 180,E1 22381.267,E2 22381.267} C_VEL
LIN {X 0,Y 291.992,Z 1051.156,A -85,B 0,C 180,E1 22390.286,E2 22390.286} C_VEL
LIN {X 0,Y 289.078,Z 1057.85,A -85,B 0,C 180,E1 22397.897,E2 22397.897} C_VEL
LIN {X 0,Y 288.189,Z 1060.787,A -85,B 0,C 180,E1 22406.987,E2 22406.987} C_VEL
LIN {X 0,Y 288.548,Z 1059.446,A -85,B 0,C 180,E1 22413.689,E2 22413.689} C_VEL
LIN {X 0,Y 290.162,Z 1053.518,A -85,B 0,C 180,E1 22422.06,E2 22422.06} C_VEL
LIN {X 0,Y 295.609,Z 1041.635,A -85,B 0,C 180,E1 22431.031,E2 22431.031} C_VEL
LIN {X 0,Y 305.883,Z 1023.327,A -85,B 0,C 180,E1 22439.699,E2 22439.699} C_VEL
LIN {X 0,Y 320.778,Z 998.641,A -85,B 0,C 180,E1 22447.463,E2 22447.463} C_VEL
LIN {X 0,Y 338.676,Z 967.987,A -85,B 0,C 180,E1 22454.022,E2 22454.022} C_VEL
LIN {X 0,Y 357.671,Z 932.236,A -85,B 0,C 180,E1 22459.252,E2 22459.252} C_VEL
LIN {X 0,Y 375.812,Z 891.829,A -85,B 0,C 180,E1 22463.337,E2 22463.337} C_VEL
LIN {X 0,Y 381.941,Z 875.992,A -85,B 0,C 180,E1 22464.565,E2 22464.565} C_VEL
LIN {X 0,Y 377.92,Z 851.981,A -85,B 0,C 180,E1 22469.248,E2 22469.248} C_VEL
LIN {X 0,Y 371.313,Z 829.088,A -85,B 0,C 180,E1 22474.751,E2 22474.751} C_VEL
LIN {X 0,Y 364.294,Z 810.938,A -85,B 0,C 180,E1 22480.558,E2 22480.558} C_VEL
LIN {X 0,Y 358.212,Z 797.055,A -85,B 0,C 180,E1 22486.921,E2 22486.921} C_VEL
LIN {X 0,Y 355.451,Z 791.007,A -85,B 0,C 180,E1 22491.305,E2 22491.305} C_VEL
LIN {X 0,Y 354.057,Z 785.256,A -85,B 0,C 180,E1 22499.382,E2 22499.382} C_VEL
LIN {X 0,Y 356.959,Z 793.072,A -85,B 0,C 180,E1 22508.079,E2 22508.079} C_VEL
LIN {X 0,Y 362.118,Z 803.886,A -85,B 0,C 180,E1 22514.073,E2 22514.073} C_VEL
LIN {X 0,Y 369.557,Z 820.667,A -85,B 0,C 180,E1 22520.175,E2 22520.175} C_VEL
LIN {X 0,Y 377.166,Z 841.12,A -85,B 0,C 180,E1 22525.584,E2 22525.584} C_VEL
LIN {X 0,Y 383.442,Z 865.451,A -85,B 0,C 180,E1 22530.581,E2 22530.581} C_VEL
LIN {X 0,Y 384.826,Z 875.66,A -85,B 0,C 180,E1 22532.296,E2 22532.296} C_VEL
LIN {X 0,Y 368.538,Z 916.774,A -85,B 0,C 180,E1 22535.443,E2 22535.443} C_VEL
LIN {X 0,Y 349.442,Z 956.734,A -85,B 0,C 180,E1 22539.911,E2 22539.911} C_VEL
LIN {X 0,Y 330.61,Z 991.249,A -85,B 0,C 180,E1 22545.555,E2 22545.555} C_VEL
LIN {X 0,Y 313.171,Z 1021.415,A -85,B 0,C 180,E1 22552.79,E2 22552.79} C_VEL
LIN {X 0,Y 299.725,Z 1045.224,A -85,B 0,C 180,E1 22561.292,E2 22561.292} C_VEL
LIN {X 0,Y 291.905,Z 1061.712,A -85,B 0,C 180,E1 22570.277,E2 22570.277} C_VEL
LIN {X 0,Y 289.051,Z 1070.536,A -85,B 0,C 180,E1 22577.893,E2 22577.893} C_VEL
LIN {X 0,Y 288.31,Z 1074.676,A -85,B 0,C 180,E1 22583.964,E2 22583.964} C_VEL
LIN {X 0,Y 288.52,Z 1076.151,A -85,B 0,C 180,E1 22589.999,E2 22589.999} C_VEL
LIN {X 0,Y 288.305,Z 1075.069,A -85,B 0,C 180,E1 22596.033,E2 22596.033} C_VEL
LIN {X 0,Y 289.413,Z 1070.351,A -85,B 0,C 180,E1 22603.488,E2 22603.488} C_VEL
LIN {X 0,Y 294.093,Z 1058.869,A -85,B 0,C 180,E1 22612.767,E2 22612.767} C_VEL
LIN {X 0,Y 303.481,Z 1041.921,A -85,B 0,C 180,E1 22621.295,E2 22621.295} C_VEL
LIN {X 0,Y 317.174,Z 1019.803,A -85,B 0,C 180,E1 22628.834,E2 22628.834} C_VEL
LIN {X 0,Y 335.445,Z 990.321,A -85,B 0,C 180,E1 22635.694,E2 22635.694} C_VEL
LIN {X 0,Y 355.031,Z 956.398,A -85,B 0,C 180,E1 22641.079,E2 22641.079} C_VEL
LIN {X 0,Y 374.489,Z 917.554,A -85,B 0,C 180,E1 22645.325,E2 22645.325} C_VEL
LIN {X 0,Y 390.442,Z 877.929,A -85,B 0,C 180,E1 22648.408,E2 22648.408} C_VEL
LIN {X 0,Y 385.086,Z 853.78,A -85,B 0,C 180,E1 22653.504,E2 22653.504} C_VEL
LIN {X 0,Y 378.623,Z 833.797,A -85,B 0,C 180,E1 22658.891,E2 22658.891} C_VEL
LIN {X 0,Y 372.385,Z 818.337,A -85,B 0,C 180,E1 22664.667,E2 22664.667} C_VEL
LIN {X 0,Y 367.651,Z 806.557,A -85,B 0,C 180,E1 22671.263,E2 22671.263} C_VEL
LIN {X 0,Y 365.629,Z 800.635,A -85,B 0,C 180,E1 22679.559,E2 22679.559} C_VEL
LIN {X 0,Y 365.413,Z 803.386,A -85,B 0,C 180,E1 22682.634,E2 22682.634} C_VEL
LIN {X 0,Y 365.011,Z 808.786,A -85,B 0,C 180,E1 22685.23,E2 22685.23} C_VEL
LIN {X 0,Y 364.75,Z 815.472,A -85,B 0,C 180,E1 22687.797,E2 22687.797} C_VEL
LIN {X 0,Y 368.494,Z 825.585,A -85,B 0,C 180,E1 22693.682,E2 22693.682} C_VEL
LIN {X 0,Y 373.549,Z 840.896,A -85,B 0,C 180,E1 22699.524,E2 22699.524} C_VEL
LIN {X 0,Y 378.303,Z 859.591,A -85,B 0,C 180,E1 22704.777,E2 22704.777} C_VEL
LIN {X 0,Y 381.881,Z 882.534,A -85,B 0,C 180,E1 22709.936,E2 22709.936} C_VEL
LIN {X 0,Y 363.836,Z 922.635,A -85,B 0,C 180,E1 22713.593,E2 22713.593} C_VEL
LIN {X 0,Y 344.432,Z 958.026,A -85,B 0,C 180,E1 22718.147,E2 22718.147} C_VEL
LIN {X 0,Y 324.164,Z 990.407,A -85,B 0,C 180,E1 22724.238,E2 22724.238} C_VEL
LIN {X 0,Y 306.573,Z 1016.549,A -85,B 0,C 180,E1 22731.525,E2 22731.525} C_VEL
LIN {X 0,Y 292.314,Z 1037.732,A -85,B 0,C 180,E1 22740.497,E2 22740.497} C_VEL
LIN {X 0,Y 284.388,Z 1051.353,A -85,B 0,C 180,E1 22749.755,E2 22749.755} C_VEL
LIN {X 0,Y 281.255,Z 1058.046,A -85,B 0,C 180,E1 22757.555,E2 22757.555} C_VEL
LIN {X 0,Y 280.28,Z 1060.995,A -85,B 0,C 180,E1 22766.902,E2 22766.902} C_VEL
LIN {X 0,Y 280.649,Z 1059.892,A -85,B 0,C 180,E1 22773.097,E2 22773.097} C_VEL
LIN {X 0,Y 281.856,Z 1055.24,A -85,B 0,C 180,E1 22780.848,E2 22780.848} C_VEL
LIN {X 0,Y 286.858,Z 1044.282,A -85,B 0,C 180,E1 22790.084,E2 22790.084} C_VEL
LIN {X 0,Y 296.742,Z 1027.086,A -85,B 0,C 180,E1 22799.023,E2 22799.023} C_VEL
LIN {X 0,Y 310.56,Z 1004.911,A -85,B 0,C 180,E1 22806.71,E2 22806.71} C_VEL
LIN {X 0,Y 327.178,Z 978.221,A -85,B 0,C 180,E1 22813.094,E2 22813.094} C_VEL
LIN {X 0,Y 346.365,Z 944.5,A -85,B 0,C 180,E1 22818.688,E2 22818.688} C_VEL
LIN {X 0,Y 365.253,Z 906.059,A -85,B 0,C 180,E1 22823.078,E2 22823.078} C_VEL
LIN {X 0,Y 376.469,Z 878.966,A -85,B 0,C 180,E1 22825.367,E2 22825.367} C_VEL
LIN {X 0,Y 372.617,Z 854.933,A -85,B 0,C 180,E1 22830.274,E2 22830.274} C_VEL
LIN {X 0,Y 366.965,Z 833.801,A -85,B 0,C 180,E1 22835.605,E2 22835.605} C_VEL
LIN {X 0,Y 360.433,Z 815.943,A -85,B 0,C 180,E1 22841.615,E2 22841.615} C_VEL
LIN {X 0,Y 355.17,Z 803.595,A -85,B 0,C 180,E1 22847.834,E2 22847.834} C_VEL
LIN {X 0,Y 353.066,Z 798.381,A -85,B 0,C 180,E1 22851.623,E2 22851.623} C_VEL
LIN {X 0,Y 352.146,Z 792.918,A -85,B 0,C 180,E1 22859.687,E2 22859.687} C_VEL
LIN {X 0,Y 354.606,Z 800.735,A -85,B 0,C 180,E1 22867.969,E2 22867.969} C_VEL
LIN {X 0,Y 359.042,Z 810.275,A -85,B 0,C 180,E1 22873.419,E2 22873.419} C_VEL
LIN {X 0,Y 365.618,Z 825.915,A -85,B 0,C 180,E1 22879.36,E2 22879.36} C_VEL
LIN {X 0,Y 372.901,Z 847.17,A -85,B 0,C 180,E1 22885.171,E2 22885.171} C_VEL
LIN {X 0,Y 378.713,Z 872.24,A -85,B 0,C 180,E1 22890.405,E2 22890.405} C_VEL
LIN {X 0,Y 379.012,Z 879.372,A -85,B 0,C 180,E1 22891.546,E2 22891.546} C_VEL
LIN {X 0,Y 362.725,Z 919.061,A -85,B 0,C 180,E1 22894.661,E2 22894.661} C_VEL
LIN {X 0,Y 343.736,Z 957.408,A -85,B 0,C 180,E1 22899.01,E2 22899.01} C_VEL
LIN {X 0,Y 324.251,Z 991.946,A -85,B 0,C 180,E1 22904.746,E2 22904.746} C_VEL
LIN {X 0,Y 307.204,Z 1020.32,A -85,B 0,C 180,E1 22911.647,E2 22911.647} C_VEL
LIN {X 0,Y 293.576,Z 1043.199,A -85,B 0,C 180,E1 22919.781,E2 22919.781} C_VEL
LIN {X 0,Y 284.783,Z 1060.302,A -85,B 0,C 180,E1 22928.963,E2 22928.963} C_VEL
LIN {X 0,Y 281.22,Z 1070.302,A -85,B 0,C 180,E1 22937.551,E2 22937.551} C_VEL
LIN {X 0,Y 280.407,Z 1074.454,A -85,B 0,C 180,E1 22943.794,E2 22943.794} C_VEL
LIN {X 0,Y 280.622,Z 1075.937,A -85,B 0,C 180,E1 22949.999,E2 22949.999} C_VEL
LIN {X 0,Y 280.398,Z 1074.866,A -85,B 0,C 180,E1 22956.204,E2 22956.204} C_VEL
LIN {X 0,Y 281.811,Z 1069.57,A -85,B 0,C 180,E1 22964.576,E2 22964.576} C_VEL
LIN {X 0,Y 287.246,Z 1057.571,A -85,B 0,C 180,E1 22974.132,E2 22974.132} C_VEL
LIN {X 0,Y 298.045,Z 1039.443,A -85,B 0,C 180,E1 22983.071,E2 22983.071} C_VEL
LIN {X 0,Y 313.192,Z 1016.031,A -85,B 0,C 180,E1 22990.782,E2 22990.782} C_VEL
LIN {X 0,Y 331.05,Z 988.174,A -85,B 0,C 180,E1 22997.087,E2 22997.087} C_VEL
LIN {X 0,Y 350.704,Z 955.057,A -85,B 0,C 180,E1 23002.268,E2 23002.268} C_VEL
LIN {X 0,Y 370.195,Z 917.045,A -85,B 0,C 180,E1 23006.391,E2 23006.391} C_VEL
LIN {X 0,Y 385.013,Z 881.133,A -85,B 0,C 180,E1 23009.23,E2 23009.23} C_VEL
LIN {X 0,Y 380.265,Z 857.865,A -85,B 0,C 180,E1 23014.376,E2 23014.376} C_VEL
LIN {X 0,Y 374.106,Z 837.913,A -85,B 0,C 180,E1 23020.058,E2 23020.058} C_VEL
LIN {X 0,Y 368.711,Z 823.844,A -85,B 0,C 180,E1 23025.728,E2 23025.728} C_VEL
LIN {X 0,Y 364.896,Z 813.857,A -85,B 0,C 180,E1 23031.647,E2 23031.647} C_VEL
LIN {X 0,Y 363.196,Z 809.327,A -85,B 0,C 180,E1 23037.613,E2 23037.613} C_VEL
LIN {X 0,Y 363.01,Z 809.619,A -85,B 0,C 180,E1 23040.901,E2 23040.901} C_VEL
LIN {X 0,Y 364.75,Z 815.472,A -85,B 0,C 180,E1 23047.797,E2 23047.797} C_VEL
LIN {X 0,Y 364.669,Z 823.145,A -85,B 0,C 180,E1 23050.28,E2 23050.28} C_VEL
LIN {X 0,Y 364.781,Z 831.227,A -85,B 0,C 180,E1 23052.748,E2 23052.748} C_VEL
LIN {X 0,Y 369.179,Z 845.502,A -85,B 0,C 180,E1 23058.557,E2 23058.557} C_VEL
LIN {X 0,Y 373.705,Z 865.013,A -85,B 0,C 180,E1 23064.245,E2 23064.245} C_VEL
LIN {X 0,Y 376.506,Z 886.266,A -85,B 0,C 180,E1 23069.214,E2 23069.214} C_VEL
LIN {X 0,Y 358.439,Z 924.501,A -85,B 0,C 180,E1 23072.72,E2 23072.72} C_VEL
LIN {X 0,Y 338.502,Z 959.631,A -85,B 0,C 180,E1 23077.315,E2 23077.315} C_VEL
LIN {X 0,Y 317.951,Z 991.321,A -85,B 0,C 180,E1 23083.38,E2 23083.38} C_VEL
LIN {X 0,Y 299.694,Z 1017.381,A -85,B 0,C 180,E1 23090.8,E2 23090.8} C_VEL
LIN {X 0,Y 285.239,Z 1037.895,A -85,B 0,C 180,E1 23099.69,E2 23099.69} C_VEL
LIN {X 0,Y 276.609,Z 1051.911,A -85,B 0,C 180,E1 23109.498,E2 23109.498} C_VEL
LIN {X 0,Y 273.431,Z 1058.242,A -85,B 0,C 180,E1 23117.193,E2 23117.193} C_VEL
LIN {X 0,Y 272.39,Z 1061.202,A -85,B 0,C 180,E1 23126.812,E2 23126.812} C_VEL
LIN {X 0,Y 272.766,Z 1060.113,A -85,B 0,C 180,E1 23133.186,E2 23133.186} C_VEL
LIN {X 0,Y 274.067,Z 1055.476,A -85,B 0,C 180,E1 23141.16,E2 23141.16} C_VEL
LIN {X 0,Y 279.342,Z 1044.542,A -85,B 0,C 180,E1 23150.649,E2 23150.649} C_VEL
LIN {X 0,Y 289.549,Z 1027.677,A -85,B 0,C 180,E1 23159.661,E2 23159.661} C_VEL
LIN {X 0,Y 304.181,Z 1005.221,A -85,B 0,C 180,E1 23167.612,E2 23167.612} C_VEL
LIN {X 0,Y 321.365,Z 978.565,A -85,B 0,C 180,E1 23174.072,E2 23174.072} C_VEL
LIN {X 0,Y 341.133,Z 944.882,A -85,B 0,C 180,E1 23179.698,E2 23179.698} C_VEL
LIN {X 0,Y 360.365,Z 906.891,A -85,B 0,C 180,E1 23184.047,E2 23184.047} C_VEL
LIN {X 0,Y 370.884,Z 882.067,A -85,B 0,C 180,E1 23186.177,E2 23186.177} C_VEL
LIN {X 0,Y 367.532,Z 858.831,A -85,B 0,C 180,E1 23191.138,E2 23191.138} C_VEL
LIN {X 0,Y 362.36,Z 838.221,A -85,B 0,C 180,E1 23196.588,E2 23196.588} C_VEL
LIN {X 0,Y 356.58,Z 821.171,A -85,B 0,C 180,E1 23202.689,E2 23202.689} C_VEL
LIN {X 0,Y 352.816,Z 811.476,A -85,B 0,C 180,E1 23207.594,E2 23207.594} C_VEL
LIN {X 0,Y 350.261,Z 805.108,A -85,B 0,C 180,E1 23212.889,E2 23212.889} C_VEL
LIN {X 0,Y 349.929,Z 800.498,A -85,B 0,C 180,E1 23219.375,E2 23219.375} C_VEL
LIN {X 0,Y 352.077,Z 807.514,A -85,B 0,C 180,E1 23227.414,E2 23227.414} C_VEL
LIN {X 0,Y 356.407,Z 818.29,A -85,B 0,C 180,E1 23233.521,E2 23233.521} C_VEL
LIN {X 0,Y 362.588,Z 834.218,A -85,B 0,C 180,E1 23239.528,E2 23239.528} C_VEL
LIN {X 0,Y 368.732,Z 853.862,A -85,B 0,C 180,E1 23244.908,E2 23244.908} C_VEL
LIN {X 0,Y 373.809,Z 878.704,A -85,B 0,C 180,E1 23250.207,E2 23250.207} C_VEL
LIN {X 0,Y 373.193,Z 883.29,A -85,B 0,C 180,E1 23250.789,E2 23250.789} C_VEL
LIN {X 0,Y 357.058,Z 920.984,A -85,B 0,C 180,E1 23253.822,E2 23253.822} C_VEL
LIN {X 0,Y 337.561,Z 959.006,A -85,B 0,C 180,E1 23258.22,E2 23258.22} C_VEL
LIN {X 0,Y 317.804,Z 992.799,A -85,B 0,C 180,E1 23263.949,E2 23263.949} C_VEL
LIN {X 0,Y 299.534,Z 1022.027,A -85,B 0,C 180,E1 23271.281,E2 23271.281} C_VEL
LIN {X 0,Y 285.537,Z 1044.68,A -85,B 0,C 180,E1 23279.721,E2 23279.721} C_VEL
LIN {X 0,Y 276.484,Z 1061.734,A -85,B 0,C 180,E1 23289.511,E2 23289.511} C_VEL
LIN {X 0,Y 273.093,Z 1071.313,A -85,B 0,C 180,E1 23298.8,E2 23298.8} C_VEL
LIN {X 0,Y 272.482,Z 1075.297,A -85,B 0,C 180,E1 23306.81,E2 23306.81} C_VEL
LIN {X 0,Y 272.562,Z 1075.507,A -85,B 0,C 180,E1 23313.186,E2 23313.186} C_VEL
LIN {X 0,Y 273.373,Z 1071.095,A -85,B 0,C 180,E1 23322.809,E2 23322.809} C_VEL
LIN {X 0,Y 277.896,Z 1060.903,A -85,B 0,C 180,E1 23332.439,E2 23332.439} C_VEL
LIN {X 0,Y 287.852,Z 1044.438,A -85,B 0,C 180,E1 23341.764,E2 23341.764} C_VEL
LIN {X 0,Y 303.817,Z 1020.746,A -85,B 0,C 180,E1 23350.421,E2 23350.421} C_VEL
LIN {X 0,Y 323.661,Z 991.137,A -85,B 0,C 180,E1 23357.557,E2 23357.557} C_VEL
LIN {X 0,Y 344.647,Z 957.076,A -85,B 0,C 180,E1 23363.06,E2 23363.06} C_VEL
LIN {X 0,Y 365.675,Z 917.342,A -85,B 0,C 180,E1 23367.408,E2 23367.408} C_VEL
LIN {X 0,Y 379.622,Z 885.765,A -85,B 0,C 180,E1 23369.846,E2 23369.846} C_VEL
LIN {X 0,Y 376.182,Z 865.516,A -85,B 0,C 180,E1 23374.344,E2 23374.344} C_VEL
LIN {X 0,Y 370.738,Z 845.502,A -85,B 0,C 180,E1 23380.07,E2 23380.07} C_VEL
LIN {X 0,Y 365.374,Z 830.492,A -85,B 0,C 180,E1 23386.208,E2 23386.208} C_VEL
LIN {X 0,Y 362.309,Z 821.596,A -85,B 0,C 180,E1 23391.587,E2 23391.587} C_VEL
LIN {X 0,Y 360.649,Z 816.874,A -85,B 0,C 180,E1 23397.596,E2 23397.596} C_VEL
LIN {X 0,Y 360.645,Z 816.337,A -85,B 0,C 180,E1 23400.004,E2 23400.004} C_VEL
LIN {X 0,Y 362.004,Z 822.639,A -85,B 0,C 180,E1 23407.537,E2 23407.537} C_VEL
LIN {X 0,Y 364.781,Z 831.227,A -85,B 0,C 180,E1 23412.748,E2 23412.748} C_VEL
LIN {X 0,Y 365.086,Z 837.483,A -85,B 0,C 180,E1 23414.559,E2 23414.559} C_VEL
LIN {X 0,Y 364.765,Z 849.888,A -85,B 0,C 180,E1 23417.443,E2 23417.443} C_VEL
LIN {X 0,Y 368.693,Z 868.823,A -85,B 0,C 180,E1 23423.308,E2 23423.308} C_VEL
LIN {X 0,Y 371.108,Z 888.851,A -85,B 0,C 180,E1 23428.218,E2 23428.218} C_VEL
LIN {X 0,Y 369.059,Z 894.679,A -85,B 0,C 180,E1 23428.823,E2 23428.823} C_VEL
LIN {X 0,Y 349.117,Z 933.901,A -85,B 0,C 180,E1 23432.686,E2 23432.686} C_VEL
LIN {X 0,Y 327.715,Z 969.07,A -85,B 0,C 180,E1 23437.765,E2 23437.765} C_VEL
LIN {X 0,Y 306.135,Z 1000.118,A -85,B 0,C 180,E1 23444.437,E2 23444.437} C_VEL
LIN {X 0,Y 288.187,Z 1024.404,A -85,B 0,C 180,E1 23452.379,E2 23452.379} C_VEL
LIN {X 0,Y 274.667,Z 1043.259,A -85,B 0,C 180,E1 23461.988,E2 23461.988} C_VEL
LIN {X 0,Y 267.434,Z 1054.852,A -85,B 0,C 180,E1 23471.843,E2 23471.843} C_VEL
LIN {X 0,Y 264.859,Z 1060.067,A -85,B 0,C 180,E1 23480.118,E2 23480.118} C_VEL
LIN {X 0,Y 264.825,Z 1061.161,A -85,B 0,C 180,E1 23490.002,E2 23490.002} C_VEL
LIN {X 0,Y 265.766,Z 1056.891,A -85,B 0,C 180,E1 23499.851,E2 23499.851} C_VEL
LIN {X 0,Y 269.967,Z 1048.154,A -85,B 0,C 180,E1 23508.832,E2 23508.832} C_VEL
LIN {X 0,Y 279.482,Z 1032.62,A -85,B 0,C 180,E1 23518.325,E2 23518.325} C_VEL
LIN {X 0,Y 293.588,Z 1011.702,A -85,B 0,C 180,E1 23526.648,E2 23526.648} C_VEL
LIN {X 0,Y 310.85,Z 986.187,A -85,B 0,C 180,E1 23533.521,E2 23533.521} C_VEL
LIN {X 0,Y 330.102,Z 955.431,A -85,B 0,C 180,E1 23539.243,E2 23539.243} C_VEL
LIN {X 0,Y 350.171,Z 918.74,A -85,B 0,C 180,E1 23543.933,E2 23543.933} C_VEL
LIN {X 0,Y 365.341,Z 884.53,A -85,B 0,C 180,E1 23547.14,E2 23547.14} C_VEL
LIN {X 0,Y 362.406,Z 861.753,A -85,B 0,C 180,E1 23552.241,E2 23552.241} C_VEL
LIN {X 0,Y 357.832,Z 842.619,A -85,B 0,C 180,E1 23557.591,E2 23557.591} C_VEL
LIN {X 0,Y 353.111,Z 827.696,A -85,B 0,C 180,E1 23563.177,E2 23563.177} C_VEL
LIN {X 0,Y 349.475,Z 817.486,A -85,B 0,C 180,E1 23568.743,E2 23568.743} C_VEL
LIN {X 0,Y 347.91,Z 812.878,A -85,B 0,C 180,E1 23572.487,E2 23572.487} C_VEL
LIN {X 0,Y 347.401,Z 808.946,A -85,B 0,C 180,E1 23577.495,E2 23577.495} C_VEL
LIN {X 0,Y 347.542,Z 808.747,A -85,B 0,C 180,E1 23579.995,E2 23579.995} C_VEL
LIN {X 0,Y 349.498,Z 815.318,A -85,B 0,C 180,E1 23587.469,E2 23587.469} C_VEL
LIN {X 0,Y 353.716,Z 826.314,A -85,B 0,C 180,E1 23593.624,E2 23593.624} C_VEL
LIN {X 0,Y 359.546,Z 842.451,A -85,B 0,C 180,E1 23599.7,E2 23599.7} C_VEL
LIN {X 0,Y 365.232,Z 864.036,A -85,B 0,C 180,E1 23605.491,E2 23605.491} C_VEL
LIN {X 0,Y 368.585,Z 883.744,A -85,B 0,C 180,E1 23609.726,E2 23609.726} C_VEL
LIN {X 0,Y 351.455,Z 922.937,A -85,B 0,C 180,E1 23612.958,E2 23612.958} C_VEL
LIN {X 0,Y 332.588,Z 958.653,A -85,B 0,C 180,E1 23617.119,E2 23617.119} C_VEL
LIN {X 0,Y 312.598,Z 991.847,A -85,B 0,C 180,E1 23622.733,E2 23622.733} C_VEL
LIN {X 0,Y 293.233,Z 1021.627,A -85,B 0,C 180,E1 23630.242,E2 23630.242} C_VEL
LIN {X 0,Y 278.507,Z 1044.405,A -85,B 0,C 180,E1 23638.873,E2 23638.873} C_VEL
LIN {X 0,Y 268.829,Z 1061.645,A -85,B 0,C 180,E1 23649.032,E2 23649.032} C_VEL
LIN {X 0,Y 265.25,Z 1071.079,A -85,B 0,C 180,E1 23658.464,E2 23658.464} C_VEL
LIN {X 0,Y 264.572,Z 1075.077,A -85,B 0,C 180,E1 23666.715,E2 23666.715} C_VEL
LIN {X 0,Y 264.648,Z 1075.298,A -85,B 0,C 180,E1 23673.281,E2 23673.281} C_VEL
LIN {X 0,Y 265.553,Z 1070.902,A -85,B 0,C 180,E1 23683.193,E2 23683.193} C_VEL
LIN {X 0,Y 270.408,Z 1060.726,A -85,B 0,C 180,E1 23693.095,E2 23693.095} C_VEL
LIN {X 0,Y 280.933,Z 1044.277,A -85,B 0,C 180,E1 23702.642,E2 23702.642} C_VEL
LIN {X 0,Y 297.674,Z 1020.611,A -85,B 0,C 180,E1 23711.436,E2 23711.436} C_VEL
LIN {X 0,Y 317.981,Z 991.407,A -85,B 0,C 180,E1 23718.564,E2 23718.564} C_VEL
LIN {X 0,Y 340.322,Z 956.229,A -85,B 0,C 180,E1 23724.248,E2 23724.248} C_VEL
LIN {X 0,Y 361.392,Z 917.315,A -85,B 0,C 180,E1 23728.486,E2 23728.486} C_VEL
LIN {X 0,Y 374.392,Z 888.488,A -85,B 0,C 180,E1 23730.78,E2 23730.78} C_VEL
LIN {X 0,Y 370.473,Z 865.965,A -85,B 0,C 180,E1 23736.181,E2 23736.181} C_VEL
LIN {X 0,Y 366.066,Z 849.415,A -85,B 0,C 180,E1 23741.354,E2 23741.354} C_VEL
LIN {X 0,Y 361.275,Z 834.787,A -85,B 0,C 180,E1 23747.898,E2 23747.898} C_VEL
LIN {X 0,Y 358.949,Z 828.106,A -85,B 0,C 180,E1 23752.728,E2 23752.728} C_VEL
LIN {X 0,Y 358.044,Z 824.398,A -85,B 0,C 180,E1 23757.579,E2 23757.579} C_VEL
LIN {X 0,Y 358.044,Z 823.861,A -85,B 0,C 180,E1 23760.004,E2 23760.004} C_VEL
LIN {X 0,Y 358.985,Z 829.757,A -85,B 0,C 180,E1 23767.28,E2 23767.28} C_VEL
LIN {X 0,Y 362.348,Z 841.158,A -85,B 0,C 180,E1 23773.919,E2 23773.919} C_VEL
LIN {X 0,Y 364.765,Z 849.888,A -85,B 0,C 180,E1 23777.443,E2 23777.443} C_VEL
LIN {X 0,Y 364.779,Z 857.119,A -85,B 0,C 180,E1 23779.162,E2 23779.162} C_VEL
LIN {X 0,Y 363.533,Z 871.018,A -85,B 0,C 180,E1 23781.88,E2 23781.88} C_VEL
LIN {X 0,Y 365.832,Z 892.635,A -85,B 0,C 180,E1 23787.445,E2 23787.445} C_VEL
LIN {X 0,Y 345.345,Z 932.998,A -85,B 0,C 180,E1 23791.446,E2 23791.446} C_VEL
LIN {X 0,Y 323.409,Z 968.141,A -85,B 0,C 180,E1 23796.445,E2 23796.445} C_VEL
LIN {X 0,Y 301.565,Z 998.71,A -85,B 0,C 180,E1 23802.93,E2 23802.93} C_VEL
LIN {X 0,Y 282.508,Z 1023.592,A -85,B 0,C 180,E1 23811.002,E2 23811.002} C_VEL
LIN {X 0,Y 268.344,Z 1042.14,A -85,B 0,C 180,E1 23820.365,E2 23820.365} C_VEL
LIN {X 0,Y 260.65,Z 1053.506,A -85,B 0,C 180,E1 23829.586,E2 23829.586} C_VEL
LIN {X 0,Y 257.826,Z 1058.635,A -85,B 0,C 180,E1 23836.404,E2 23836.404} C_VEL
LIN {X 0,Y 256.584,Z 1061.618,A -85,B 0,C 180,E1 23846.616,E2 23846.616} C_VEL
LIN {X 0,Y 256.969,Z 1060.556,A -85,B 0,C 180,E1 23853.382,E2 23853.382} C_VEL
LIN {X 0,Y 258.485,Z 1055.949,A -85,B 0,C 180,E1 23861.842,E2 23861.842} C_VEL
LIN {X 0,Y 264.437,Z 1045.062,A -85,B 0,C 180,E1 23871.871,E2 23871.871} C_VEL
LIN {X 0,Y 275.874,Z 1027.99,A -85,B 0,C 180,E1 23881.43,E2 23881.43} C_VEL
LIN {X 0,Y 291.644,Z 1005.843,A -85,B 0,C 180,E1 23889.534,E2 23889.534} C_VEL
LIN {X 0,Y 310.023,Z 979.25,A -85,B 0,C 180,E1 23896.138,E2 23896.138} C_VEL
LIN {X 0,Y 331.323,Z 945.093,A -85,B 0,C 180,E1 23901.882,E2 23901.882} C_VEL
LIN {X 0,Y 351.899,Z 906.386,A -85,B 0,C 180,E1 23906.272,E2 23906.272} C_VEL
LIN {X 0,Y 359.637,Z 889.267,A -85,B 0,C 180,E1 23907.761,E2 23907.761} C_VEL
LIN {X 0,Y 358.169,Z 870.709,A -85,B 0,C 180,E1 23911.884,E2 23911.884} C_VEL
LIN {X 0,Y 354.403,Z 850.963,A -85,B 0,C 180,E1 23917.362,E2 23917.362} C_VEL
LIN {X 0,Y 349.681,Z 834.188,A -85,B 0,C 180,E1 23923.676,E2 23923.676} C_VEL
LIN {X 0,Y 346.259,Z 823.273,A -85,B 0,C 180,E1 23929.913,E2 23929.913} C_VEL
LIN {X 0,Y 344.836,Z 816.539,A -85,B 0,C 180,E1 23937.477,E2 23937.477} C_VEL
LIN {X 0,Y 344.977,Z 816.337,A -85,B 0,C 180,E1 23939.995,E2 23939.995} C_VEL
LIN {X 0,Y 346.897,Z 823.079,A -85,B 0,C 180,E1 23947.526,E2 23947.526} C_VEL
LIN {X 0,Y 350.753,Z 834.148,A -85,B 0,C 180,E1 23953.741,E2 23953.741} C_VEL
LIN {X 0,Y 356.101,Z 850.729,A -85,B 0,C 180,E1 23959.899,E2 23959.899} C_VEL
LIN {X 0,Y 360.962,Z 871.618,A -85,B 0,C 180,E1 23965.483,E2 23965.483} C_VEL
LIN {X 0,Y 363.014,Z 887.927,A -85,B 0,C 180,E1 23968.986,E2 23968.986} C_VEL
LIN {X 0,Y 344.277,Z 928.243,A -85,B 0,C 180,E1 23972.402,E2 23972.402} C_VEL
LIN {X 0,Y 324.252,Z 964.137,A -85,B 0,C 180,E1 23976.835,E2 23976.835} C_VEL
LIN {X 0,Y 304.907,Z 994.804,A -85,B 0,C 180,E1 23982.327,E2 23982.327} C_VEL
LIN {X 0,Y 286.179,Z 1022.437,A -85,B 0,C 180,E1 23989.557,E2 23989.557} C_VEL
LIN {X 0,Y 271.545,Z 1044.129,A -85,B 0,C 180,E1 23997.982,E2 23997.982} C_VEL
LIN {X 0,Y 261.532,Z 1060.812,A -85,B 0,C 180,E1 24007.968,E2 24007.968} C_VEL
LIN {X 0,Y 257.413,Z 1070.845,A -85,B 0,C 180,E1 24018.108,E2 24018.108} C_VEL
LIN {X 0,Y 256.677,Z 1074.858,A -85,B 0,C 180,E1 24026.614,E2 24026.614} C_VEL
LIN {X 0,Y 256.76,Z 1075.09,A -85,B 0,C 180,E1 24033.382,E2 24033.382} C_VEL
LIN {X 0,Y 257.768,Z 1070.709,A -85,B 0,C 180,E1 24043.599,E2 24043.599} C_VEL
LIN {X 0,Y 262.97,Z 1060.55,A -85,B 0,C 180,E1 24053.788,E2 24053.788} C_VEL
LIN {X 0,Y 274.096,Z 1044.116,A -85,B 0,C 180,E1 24063.562,E2 24063.562} C_VEL
LIN {X 0,Y 291.593,Z 1020.474,A -85,B 0,C 180,E1 24072.499,E2 24072.499} C_VEL
LIN {X 0,Y 312.255,Z 991.849,A -85,B 0,C 180,E1 24079.567,E2 24079.567} C_VEL
LIN {X 0,Y 335.297,Z 956.745,A -85,B 0,C 180,E1 24085.292,E2 24085.292} C_VEL
LIN {X 0,Y 357.463,Z 916.946,A -85,B 0,C 180,E1 24089.606,E2 24089.606} C_VEL
LIN {X 0,Y 368.865,Z 892.651,A -85,B 0,C 180,E1 24091.514,E2 24091.514} C_VEL
LIN {X 0,Y 366.429,Z 873.749,A -85,B 0,C 180,E1 24096.099,E2 24096.099} C_VEL
LIN {X 0,Y 362.271,Z 855.927,A -85,B 0,C 180,E1 24101.721,E2 24101.721} C_VEL
LIN {X 0,Y 358.231,Z 842.511,A -85,B 0,C 180,E1 24107.794,E2 24107.794} C_VEL
LIN {X 0,Y 356.069,Z 835.566,A -85,B 0,C 180,E1 24112.669,E2 24112.669} C_VEL
LIN {X 0,Y 355.156,Z 831.824,A -85,B 0,C 180,E1 24117.559,E2 24117.559} C_VEL
LIN {X 0,Y 355.158,Z 831.277,A -85,B 0,C 180,E1 24120.004,E2 24120.004} C_VEL
LIN {X 0,Y 356.052,Z 837.326,A -85,B 0,C 180,E1 24127.34,E2 24127.34} C_VEL
LIN {X 0,Y 358.881,Z 848.309,A -85,B 0,C 180,E1 24133.792,E2 24133.792} C_VEL
LIN {X 0,Y 362.252,Z 863.469,A -85,B 0,C 180,E1 24139.556,E2 24139.556} C_VEL
LIN {X 0,Y 363.533,Z 871.018,A -85,B 0,C 180,E1 24141.88,E2 24141.88} C_VEL
LIN {X 0,Y 362.949,Z 879.181,A -85,B 0,C 180,E1 24143.498,E2 24143.498} C_VEL
LIN {X 0,Y 360.415,Z 894.061,A -85,B 0,C 180,E1 24146.074,E2 24146.074} C_VEL
LIN {X 0,Y 359.803,Z 898.213,A -85,B 0,C 180,E1 24146.881,E2 24146.881} C_VEL
LIN {X 0,Y 339.85,Z 935.305,A -85,B 0,C 180,E1 24150.557,E2 24150.557} C_VEL
LIN {X 0,Y 317.094,Z 970.502,A -85,B 0,C 180,E1 24155.668,E2 24155.668} C_VEL
LIN {X 0,Y 294.877,Z 1000.391,A -85,B 0,C 180,E1 24162.176,E2 24162.176} C_VEL
LIN {X 0,Y 275.206,Z 1025.012,A -85,B 0,C 180,E1 24170.443,E2 24170.443} C_VEL
LIN {X 0,Y 260.625,Z 1043.225,A -85,B 0,C 180,E1 24180.069,E2 24180.069} C_VEL
LIN {X 0,Y 252.149,Z 1055.219,A -85,B 0,C 180,E1 24190.7,E2 24190.7} C_VEL
LIN {X 0,Y 249.157,Z 1060.472,A -85,B 0,C 180,E1 24199.488,E2 24199.488} C_VEL
LIN {X 0,Y 249.029,Z 1061.589,A -85,B 0,C 180,E1 24210.002,E2 24210.002} C_VEL
LIN {X 0,Y 250.121,Z 1057.363,A -85,B 0,C 180,E1 24220.474,E2 24220.474} C_VEL
LIN {X 0,Y 254.885,Z 1048.661,A -85,B 0,C 180,E1 24229.992,E2 24229.992} C_VEL
LIN {X 0,Y 266.646,Z 1031.631,A -85,B 0,C 180,E1 24240.765,E2 24240.765} C_VEL
LIN {X 0,Y 283.763,Z 1008.521,A -85,B 0,C 180,E1 24249.857,E2 24249.857} C_VEL
LIN {X 0,Y 304.51,Z 979.592,A -85,B 0,C 180,E1 24257.228,E2 24257.228} C_VEL
LIN {X 0,Y 326.183,Z 945.961,A -85,B 0,C 180,E1 24262.917,E2 24262.917} C_VEL
LIN {X 0,Y 347.54,Z 906.818,A -85,B 0,C 180,E1 24267.364,E2 24267.364} C_VEL
LIN {X 0,Y 354.528,Z 891.51,A -85,B 0,C 180,E1 24268.749,E2 24268.749} C_VEL
LIN {X 0,Y 352.412,Z 869.216,A -85,B 0,C 180,E1 24274.185,E2 24274.185} C_VEL
LIN {X 0,Y 348.672,Z 850.32,A -85,B 0,C 180,E1 24280.146,E2 24280.146} C_VEL
LIN {X 0,Y 345.21,Z 837.488,A -85,B 0,C 180,E1 24285.781,E2 24285.781} C_VEL
LIN {X 0,Y 342.563,Z 827.913,A -85,B 0,C 180,E1 24292.369,E2 24292.369} C_VEL
LIN {X 0,Y 342.219,Z 824.074,A -85,B 0,C 180,E1 24297.457,E2 24297.457} C_VEL
LIN {X 0,Y 342.378,Z 823.897,A -85,B 0,C 180,E1 24299.995,E2 24299.995} C_VEL
LIN {X 0,Y 344.022,Z 830.684,A -85,B 0,C 180,E1 24307.589,E2 24307.589} C_VEL
LIN {X 0,Y 348.189,Z 843.348,A -85,B 0,C 180,E1 24314.488,E2 24314.488} C_VEL
LIN {X 0,Y 353.017,Z 860.838,A -85,B 0,C 180,E1 24320.674,E2 24320.674} C_VEL
LIN {X 0,Y 356.848,Z 882.086,A -85,B 0,C 180,E1 24326.193,E2 24326.193} C_VEL
LIN {X 0,Y 357.139,Z 892.142,A -85,B 0,C 180,E1 24328.197,E2 24328.197} C_VEL
LIN {X 0,Y 338.119,Z 931.47,A -85,B 0,C 180,E1 24331.617,E2 24331.617} C_VEL
LIN {X 0,Y 317.134,Z 967.634,A -85,B 0,C 180,E1 24336.244,E2 24336.244} C_VEL
LIN {X 0,Y 295.101,Z 1000.837,A -85,B 0,C 180,E1 24342.578,E2 24342.578} C_VEL
LIN {X 0,Y 275.41,Z 1028.564,A -85,B 0,C 180,E1 24350.644,E2 24350.644} C_VEL
LIN {X 0,Y 260.746,Z 1049.548,A -85,B 0,C 180,E1 24360.032,E2 24360.032} C_VEL
LIN {X 0,Y 251.98,Z 1064.502,A -85,B 0,C 180,E1 24370.683,E2 24370.683} C_VEL
LIN {X 0,Y 249.255,Z 1071.791,A -85,B 0,C 180,E1 24379.489,E2 24379.489} C_VEL
LIN {X 0,Y 248.766,Z 1074.637,A -85,B 0,C 180,E1 24386.506,E2 24386.506} C_VEL
LIN {X 0,Y 248.845,Z 1074.881,A -85,B 0,C 180,E1 24393.49,E2 24393.49} C_VEL
LIN {X 0,Y 249.994,Z 1070.516,A -85,B 0,C 180,E1 24404.031,E2 24404.031} C_VEL
LIN {X 0,Y 255.545,Z 1060.373,A -85,B 0,C 180,E1 24414.524,E2 24414.524} C_VEL
LIN {X 0,Y 267.329,Z 1043.954,A -85,B 0,C 180,E1 24424.53,E2 24424.53} C_VEL
LIN {X 0,Y 285.634,Z 1020.337,A -85,B 0,C 180,E1 24433.604,E2 24433.604} C_VEL
LIN {X 0,Y 307.761,Z 990.826,A -85,B 0,C 180,E1 24440.901,E2 24440.901} C_VEL
LIN {X 0,Y 330.815,Z 956.552,A -85,B 0,C 180,E1 24446.464,E2 24446.464} C_VEL
LIN {X 0,Y 353.157,Z 917.517,A -85,B 0,C 180,E1 24450.672,E2 24450.672} C_VEL
LIN {X 0,Y 363.566,Z 896.064,A -85,B 0,C 180,E1 24452.371,E2 24452.371} C_VEL
LIN {X 0,Y 361.31,Z 876.716,A -85,B 0,C 180,E1 24457.324,E2 24457.324} C_VEL
LIN {X 0,Y 357.847,Z 860.562,A -85,B 0,C 180,E1 24462.761,E2 24462.761} C_VEL
LIN {X 0,Y 354.399,Z 847.917,A -85,B 0,C 180,E1 24468.912,E2 24468.912} C_VEL
LIN {X 0,Y 353.03,Z 842.988,A -85,B 0,C 180,E1 24472.606,E2 24472.606} C_VEL
LIN {X 0,Y 352.253,Z 839.234,A -85,B 0,C 180,E1 24477.539,E2 24477.539} C_VEL
LIN {X 0,Y 352.263,Z 838.675,A -85,B 0,C 180,E1 24480.004,E2 24480.004} C_VEL
LIN {X 0,Y 352.79,Z 844.776,A -85,B 0,C 180,E1 24487.408,E2 24487.408} C_VEL
LIN {X 0,Y 355.355,Z 855.975,A -85,B 0,C 180,E1 24493.931,E2 24493.931} C_VEL
LIN {X 0,Y 358.216,Z 871.428,A -85,B 0,C 180,E1 24499.786,E2 24499.786} C_VEL
LIN {X 0,Y 360.263,Z 891.374,A -85,B 0,C 180,E1 24505.412,E2 24505.412} C_VEL
LIN {X 0,Y 360.415,Z 894.061,A -85,B 0,C 180,E1 24506.074,E2 24506.074} C_VEL
LIN {X 0,Y 358.216,Z 899.387,A -85,B 0,C 180,E1 24506.652,E2 24506.652} C_VEL
LIN {X 0,Y 348.273,Z 913.482,A -85,B 0,C 180,E1 24507.058,E2 24507.058} C_VEL
LIN {X 0,Y 326.83,Z 949.436,A -85,B 0,C 180,E1 24511.147,E2 24511.147} C_VEL
LIN {X 0,Y 304.241,Z 981.672,A -85,B 0,C 180,E1 24516.568,E2 24516.568} C_VEL
LIN {X 0,Y 282.312,Z 1009.317,A -85,B 0,C 180,E1 24523.562,E2 24523.562} C_VEL
LIN {X 0,Y 262.612,Z 1032.489,A -85,B 0,C 180,E1 24532.708,E2 24532.708} C_VEL
LIN {X 0,Y 249.652,Z 1048.364,A -85,B 0,C 180,E1 24542.921,E2 24542.921} C_VEL
LIN {X 0,Y 242.858,Z 1057.946,A -85,B 0,C 180,E1 24553.694,E2 24553.694} C_VEL
LIN {X 0,Y 240.804,Z 1061.667,A -85,B 0,C 180,E1 24562.771,E2 24562.771} C_VEL
LIN {X 0,Y 241.135,Z 1061.803,A -85,B 0,C 180,E1 24570.002,E2 24570.002} C_VEL
LIN {X 0,Y 242.313,Z 1057.599,A -85,B 0,C 180,E1 24580.815,E2 24580.815} C_VEL
LIN {X 0,Y 247.389,Z 1048.913,A -85,B 0,C 180,E1 24590.625,E2 24590.625} C_VEL
LIN {X 0,Y 259.763,Z 1031.916,A -85,B 0,C 180,E1 24601.673,E2 24601.673} C_VEL
LIN {X 0,Y 277.67,Z 1008.83,A -85,B 0,C 180,E1 24610.914,E2 24610.914} C_VEL
LIN {X 0,Y 299.105,Z 979.935,A -85,B 0,C 180,E1 24618.359,E2 24618.359} C_VEL
LIN {X 0,Y 321.446,Z 946.331,A -85,B 0,C 180,E1 24624.05,E2 24624.05} C_VEL
LIN {X 0,Y 343.366,Z 907.138,A -85,B 0,C 180,E1 24628.493,E2 24628.493} C_VEL
LIN {X 0,Y 348.991,Z 895.49,A -85,B 0,C 180,E1 24629.521,E2 24629.521} C_VEL
LIN {X 0,Y 347.939,Z 876.62,A -85,B 0,C 180,E1 24634.176,E2 24634.176} C_VEL
LIN {X 0,Y 344.886,Z 857.865,A -85,B 0,C 180,E1 24640.086,E2 24640.086} C_VEL
LIN {X 0,Y 341.923,Z 845.154,A -85,B 0,C 180,E1 24645.642,E2 24645.642} C_VEL
LIN {X 0,Y 339.87,Z 836.311,A -85,B 0,C 180,E1 24651.481,E2 24651.481} C_VEL
LIN {X 0,Y 339.331,Z 831.498,A -85,B 0,C 180,E1 24657.436,E2 24657.436} C_VEL
LIN {X 0,Y 339.475,Z 831.354,A -85,B 0,C 180,E1 24659.995,E2 24659.995} C_VEL
LIN {X 0,Y 340.84,Z 837.208,A -85,B 0,C 180,E1 24666.932,E2 24666.932} C_VEL
LIN {X 0,Y 344.513,Z 849.977,A -85,B 0,C 180,E1 24674.125,E2 24674.125} C_VEL
LIN {X 0,Y 348.75,Z 867.204,A -85,B 0,C 180,E1 24680.337,E2 24680.337} C_VEL
LIN {X 0,Y 352.022,Z 888.537,A -85,B 0,C 180,E1 24685.965,E2 24685.965} C_VEL
LIN {X 0,Y 352.346,Z 894.026,A -85,B 0,C 180,E1 24687.215,E2 24687.215} C_VEL
LIN {X 0,Y 333.276,Z 932.256,A -85,B 0,C 180,E1 24690.559,E2 24690.559} C_VEL
LIN {X 0,Y 311.826,Z 968.202,A -85,B 0,C 180,E1 24695.181,E2 24695.181} C_VEL
LIN {X 0,Y 288.547,Z 1002.008,A -85,B 0,C 180,E1 24701.742,E2 24701.742} C_VEL
LIN {X 0,Y 268.782,Z 1028.738,A -85,B 0,C 180,E1 24709.705,E2 24709.705} C_VEL
LIN {X 0,Y 253.07,Z 1050.217,A -85,B 0,C 180,E1 24719.631,E2 24719.631} C_VEL
LIN {X 0,Y 244.35,Z 1064.252,A -85,B 0,C 180,E1 24730.055,E2 24730.055} C_VEL
LIN {X 0,Y 241.425,Z 1071.564,A -85,B 0,C 180,E1 24739.144,E2 24739.144} C_VEL
LIN {X 0,Y 240.854,Z 1074.417,A -85,B 0,C 180,E1 24746.391,E2 24746.391} C_VEL
LIN {X 0,Y 240.954,Z 1074.673,A -85,B 0,C 180,E1 24753.604,E2 24753.604} C_VEL
LIN {X 0,Y 242.206,Z 1070.322,A -85,B 0,C 180,E1 24764.492,E2 24764.492} C_VEL
LIN {X 0,Y 248.187,Z 1060.196,A -85,B 0,C 180,E1 24775.302,E2 24775.302} C_VEL
LIN {X 0,Y 260.655,Z 1043.792,A -85,B 0,C 180,E1 24785.546,E2 24785.546} C_VEL
LIN {X 0,Y 279.773,Z 1020.199,A -85,B 0,C 180,E1 24794.759,E2 24794.759} C_VEL
LIN {X 0,Y 302.614,Z 990.854,A -85,B 0,C 180,E1 24802.063,E2 24802.063} C_VEL
LIN {X 0,Y 326.421,Z 956.474,A -85,B 0,C 180,E1 24807.646,E2 24807.646} C_VEL
LIN {X 0,Y 349.253,Z 917.598,A -85,B 0,C 180,E1 24811.804,E2 24811.804} C_VEL
LIN {X 0,Y 358.412,Z 899.326,A -85,B 0,C 180,E1 24813.266,E2 24813.266} C_VEL
LIN {X 0,Y 356.174,Z 879.099,A -85,B 0,C 180,E1 24818.805,E2 24818.805} C_VEL
LIN {X 0,Y 353.115,Z 863.844,A -85,B 0,C 180,E1 24824.446,E2 24824.446} C_VEL
LIN {X 0,Y 350.177,Z 851.825,A -85,B 0,C 180,E1 24831.293,E2 24831.293} C_VEL
LIN {X 0,Y 349.032,Z 846.526,A -85,B 0,C 180,E1 24837.516,E2 24837.516} C_VEL
LIN {X 0,Y 349.042,Z 845.965,A -85,B 0,C 180,E1 24840.005,E2 24840.005} C_VEL
LIN {X 0,Y 349.531,Z 852.206,A -85,B 0,C 180,E1 24847.478,E2 24847.478} C_VEL
LIN {X 0,Y 351.528,Z 862.798,A -85,B 0,C 180,E1 24853.72,E2 24853.72} C_VEL
LIN {X 0,Y 353.838,Z 878.054,A -85,B 0,C 180,E1 24859.578,E2 24859.578} C_VEL
LIN {X 0,Y 355.14,Z 897.841,A -85,B 0,C 180,E1 24865.263,E2 24865.263} C_VEL
LIN {X 0,Y 354.254,Z 902.175,A -85,B 0,C 180,E1 24866.065,E2 24866.065} C_VEL
LIN {X 0,Y 348.273,Z 913.482,A -85,B 0,C 180,E1 24867.058,E2 24867.058} C_VEL
LIN {X 0,Y 338.567,Z 927.344,A -85,B 0,C 180,E1 24867.854,E2 24867.854} C_VEL
LIN {X 0,Y 328.551,Z 940.604,A -85,B 0,C 180,E1 24868.782,E2 24868.782} C_VEL
LIN {X 0,Y 306.674,Z 972.274,A -85,B 0,C 180,E1 24873.505,E2 24873.505} C_VEL
LIN {X 0,Y 283.921,Z 1000.957,A -85,B 0,C 180,E1 24879.835,E2 24879.835} C_VEL
LIN {X 0,Y 263.161,Z 1024.918,A -85,B 0,C 180,E1 24888.027,E2 24888.027} C_VEL
LIN {X 0,Y 246.252,Z 1043.983,A -85,B 0,C 180,E1 24898.463,E2 24898.463} C_VEL
LIN {X 0,Y 236.928,Z 1055.588,A -85,B 0,C 180,E1 24909.406,E2 24909.406} C_VEL
LIN {X 0,Y 233.487,Z 1060.876,A -85,B 0,C 180,E1 24918.774,E2 24918.774} C_VEL
LIN {X 0,Y 233.227,Z 1062.018,A -85,B 0,C 180,E1 24930.002,E2 24930.002} C_VEL
LIN {X 0,Y 233.707,Z 1059.828,A -85,B 0,C 180,E1 24937.453,E2 24937.453} C_VEL
LIN {X 0,Y 237.116,Z 1053.418,A -85,B 0,C 180,E1 24947.07,E2 24947.07} C_VEL
LIN {X 0,Y 247.016,Z 1039.587,A -85,B 0,C 180,E1 24958.39,E2 24958.39} C_VEL
LIN {X 0,Y 261.44,Z 1021.557,A -85,B 0,C 180,E1 24967.491,E2 24967.491} C_VEL
LIN {X 0,Y 280.786,Z 997.484,A -85,B 0,C 180,E1 24975.437,E2 24975.437} C_VEL
LIN {X 0,Y 301.847,Z 969.151,A -85,B 0,C 180,E1 24981.671,E2 24981.671} C_VEL
LIN {X 0,Y 324.645,Z 933.958,A -85,B 0,C 180,E1 24986.858,E2 24986.858} C_VEL
LIN {X 0,Y 343.797,Z 897.64,A -85,B 0,C 180,E1 24990.631,E2 24990.631} C_VEL
LIN {X 0,Y 342.61,Z 876.671,A -85,B 0,C 180,E1 24996.26,E2 24996.26} C_VEL
LIN {X 0,Y 339.872,Z 859.145,A -85,B 0,C 180,E1 25002.48,E2 25002.48} C_VEL
LIN {X 0,Y 337.538,Z 847.795,A -85,B 0,C 180,E1 25008.338,E2 25008.338} C_VEL
LIN {X 0,Y 336.53,Z 842.834,A -85,B 0,C 180,E1 25012.232,E2 25012.232} C_VEL
LIN {X 0,Y 336.411,Z 838.931,A -85,B 0,C 180,E1 25017.414,E2 25017.414} C_VEL
LIN {X 0,Y 336.566,Z 838.802,A -85,B 0,C 180,E1 25019.995,E2 25019.995} C_VEL
LIN {X 0,Y 337.682,Z 844.721,A -85,B 0,C 180,E1 25026.998,E2 25026.998} C_VEL
LIN {X 0,Y 340.729,Z 856.18,A -85,B 0,C 180,E1 25033.564,E2 25033.564} C_VEL
LIN {X 0,Y 344.423,Z 873.338,A -85,B 0,C 180,E1 25039.932,E2 25039.932} C_VEL
LIN {X 0,Y 346.851,Z 893.637,A -85,B 0,C 180,E1 25045.455,E2 25045.455} C_VEL
LIN {X 0,Y 346.651,Z 898.044,A -85,B 0,C 180,E1 25046.354,E2 25046.354} C_VEL
LIN {X 0,Y 327.196,Z 935.372,A -85,B 0,C 180,E1 25049.724,E2 25049.724} C_VEL
LIN {X 0,Y 305.811,Z 969.876,A -85,B 0,C 180,E1 25054.266,E2 25054.266} C_VEL
LIN {X 0,Y 282.822,Z 1002.15,A -85,B 0,C 180,E1 25060.625,E2 25060.625} C_VEL
LIN {X 0,Y 262.359,Z 1028.732,A -85,B 0,C 180,E1 25068.657,E2 25068.657} C_VEL
LIN {X 0,Y 246.314,Z 1049.595,A -85,B 0,C 180,E1 25078.468,E2 25078.468} C_VEL
LIN {X 0,Y 236.767,Z 1064.003,A -85,B 0,C 180,E1 25089.387,E2 25089.387} C_VEL
LIN {X 0,Y 233.574,Z 1071.336,A -85,B 0,C 180,E1 25098.775,E2 25098.775} C_VEL
LIN {X 0,Y 232.943,Z 1074.197,A -85,B 0,C 180,E1 25106.268,E2 25106.268} C_VEL
LIN {X 0,Y 233.037,Z 1074.464,A -85,B 0,C 180,E1 25113.727,E2 25113.727} C_VEL
LIN {X 0,Y 234.437,Z 1070.129,A -85,B 0,C 180,E1 25124.983,E2 25124.983} C_VEL
LIN {X 0,Y 240.86,Z 1060.019,A -85,B 0,C 180,E1 25136.128,E2 25136.128} C_VEL
LIN {X 0,Y 254.059,Z 1043.628,A -85,B 0,C 180,E1 25146.616,E2 25146.616} C_VEL
LIN {X 0,Y 274.046,Z 1020.06,A -85,B 0,C 180,E1 25155.959,E2 25155.959} C_VEL
LIN {X 0,Y 297.677,Z 990.743,A -85,B 0,C 180,E1 25163.299,E2 25163.299} C_VEL
LIN {X 0,Y 322.72,Z 955.589,A -85,B 0,C 180,E1 25168.964,E2 25168.964} C_VEL
LIN {X 0,Y 346.264,Z 916.282,A -85,B 0,C 180,E1 25173.085,E2 25173.085} C_VEL
LIN {X 0,Y 353.245,Z 902.355,A -85,B 0,C 180,E1 25174.272,E2 25174.272} C_VEL
LIN {X 0,Y 351.4,Z 883.172,A -85,B 0,C 180,E1 25179.823,E2 25179.823} C_VEL
LIN {X 0,Y 348.726,Z 868.522,A -85,B 0,C 180,E1 25185.679,E2 25185.679} C_VEL
LIN {X 0,Y 346.744,Z 859.196,A -85,B 0,C 180,E1 25191.206,E2 25191.206} C_VEL
LIN {X 0,Y 345.818,Z 853.798,A -85,B 0,C 180,E1 25197.493,E2 25197.493} C_VEL
LIN {X 0,Y 345.821,Z 853.248,A -85,B 0,C 180,E1 25200.005,E2 25200.005} C_VEL
LIN {X 0,Y 345.956,Z 859.507,A -85,B 0,C 180,E1 25207.556,E2 25207.556} C_VEL
LIN {X 0,Y 347.643,Z 870.017,A -85,B 0,C 180,E1 25213.725,E2 25213.725} C_VEL
LIN {X 0,Y 349.288,Z 884.414,A -85,B 0,C 180,E1 25219.323,E2 25219.323} C_VEL
LIN {X 0,Y 349.923,Z 903.063,A -85,B 0,C 180,E1 25224.813,E2 25224.813} C_VEL
LIN {X 0,Y 340.139,Z 921.645,A -85,B 0,C 180,E1 25226.638,E2 25226.638} C_VEL
LIN {X 0,Y 328.551,Z 940.604,A -85,B 0,C 180,E1 25228.782,E2 25228.782} C_VEL
LIN {X 0,Y 318.067,Z 953.383,A -85,B 0,C 180,E1 25229.836,E2 25229.836} C_VEL
LIN {X 0,Y 307.317,Z 965.526,A -85,B 0,C 180,E1 25231.036,E2 25231.036} C_VEL
LIN {X 0,Y 284.25,Z 994.623,A -85,B 0,C 180,E1 25236.903,E2 25236.903} C_VEL
LIN {X 0,Y 262.451,Z 1019.185,A -85,B 0,C 180,E1 25244.399,E2 25244.399} C_VEL
LIN {X 0,Y 244.432,Z 1038.577,A -85,B 0,C 180,E1 25253.713,E2 25253.713} C_VEL
LIN {X 0,Y 231.982,Z 1052.572,A -85,B 0,C 180,E1 25264.876,E2 25264.876} C_VEL
LIN {X 0,Y 226.776,Z 1059.422,A -85,B 0,C 180,E1 25274.499,E2 25274.499} C_VEL
LIN {X 0,Y 224.947,Z 1062.45,A -85,B 0,C 180,E1 25286.139,E2 25286.139} C_VEL
LIN {X 0,Y 225.388,Z 1061.441,A -85,B 0,C 180,E1 25293.857,E2 25293.857} C_VEL
LIN {X 0,Y 228.275,Z 1055.469,A -85,B 0,C 180,E1 25305.401,E2 25305.401} C_VEL
LIN {X 0,Y 236.812,Z 1043.78,A -85,B 0,C 180,E1 25316.614,E2 25316.614} C_VEL
LIN {X 0,Y 251.936,Z 1025.667,A -85,B 0,C 180,E1 25326.979,E2 25326.979} C_VEL
LIN {X 0,Y 272.525,Z 1001.172,A -85,B 0,C 180,E1 25335.721,E2 25335.721} C_VEL
LIN {X 0,Y 295.758,Z 971.145,A -85,B 0,C 180,E1 25342.581,E2 25342.581} C_VEL
LIN {X 0,Y 319.696,Z 935.402,A -85,B 0,C 180,E1 25347.921,E2 25347.921} C_VEL
LIN {X 0,Y 338.414,Z 901.859,A -85,B 0,C 180,E1 25351.346,E2 25351.346} C_VEL
LIN {X 0,Y 337.926,Z 881.891,A -85,B 0,C 180,E1 25356.892,E2 25356.892} C_VEL
LIN {X 0,Y 335.9,Z 865.422,A -85,B 0,C 180,E1 25362.927,E2 25362.927} C_VEL
LIN {X 0,Y 333.81,Z 853.437,A -85,B 0,C 180,E1 25369.533,E2 25369.533} C_VEL
LIN {X 0,Y 332.925,Z 848.15,A -85,B 0,C 180,E1 25374.772,E2 25374.772} C_VEL
LIN {X 0,Y 333.19,Z 846.221,A -85,B 0,C 180,E1 25377.388,E2 25377.388} C_VEL
LIN {X 0,Y 333.167,Z 847.201,A -85,B 0,C 180,E1 25381.298,E2 25381.298} C_VEL
LIN {X 0,Y 334.418,Z 852.155,A -85,B 0,C 180,E1 25387.066,E2 25387.066} C_VEL
LIN {X 0,Y 337.018,Z 863.672,A -85,B 0,C 180,E1 25393.649,E2 25393.649} C_VEL
LIN {X 0,Y 339.892,Z 879.344,A -85,B 0,C 180,E1 25399.531,E2 25399.531} C_VEL
LIN {X 0,Y 341.732,Z 899.091,A -85,B 0,C 180,E1 25405.02,E2 25405.02} C_VEL
LIN {X 0,Y 340.478,Z 903.162,A -85,B 0,C 180,E1 25405.551,E2 25405.551} C_VEL
LIN {X 0,Y 317.835,Z 944.219,A -85,B 0,C 180,E1 25409.523,E2 25409.523} C_VEL
LIN {X 0,Y 294.563,Z 979.164,A -85,B 0,C 180,E1 25414.598,E2 25414.598} C_VEL
LIN {X 0,Y 270.958,Z 1010.364,A -85,B 0,C 180,E1 25421.578,E2 25421.578} C_VEL
LIN {X 0,Y 250.161,Z 1035.888,A -85,B 0,C 180,E1 25430.499,E2 25430.499} C_VEL
LIN {X 0,Y 234.977,Z 1055.123,A -85,B 0,C 180,E1 25441.276,E2 25441.276} C_VEL
LIN {X 0,Y 227.354,Z 1067.163,A -85,B 0,C 180,E1 25452.544,E2 25452.544} C_VEL
LIN {X 0,Y 225.171,Z 1072.882,A -85,B 0,C 180,E1 25462.263,E2 25462.263} C_VEL
LIN {X 0,Y 225.373,Z 1074.442,A -85,B 0,C 180,E1 25469.998,E2 25469.998} C_VEL
LIN {X 0,Y 225.148,Z 1073.441,A -85,B 0,C 180,E1 25477.734,E2 25477.734} C_VEL
LIN {X 0,Y 227.378,Z 1068.686,A -85,B 0,C 180,E1 25487.45,E2 25487.45} C_VEL
LIN {X 0,Y 235.346,Z 1057.584,A -85,B 0,C 180,E1 25498.801,E2 25498.801} C_VEL
LIN {X 0,Y 249.022,Z 1041.745,A -85,B 0,C 180,E1 25508.589,E2 25508.589} C_VEL
LIN {X 0,Y 269.374,Z 1018.826,A -85,B 0,C 180,E1 25517.549,E2 25517.549} C_VEL
LIN {X 0,Y 294.077,Z 989.062,A -85,B 0,C 180,E1 25524.888,E2 25524.888} C_VEL
LIN {X 0,Y 319.642,Z 953.961,A -85,B 0,C 180,E1 25530.402,E2 25530.402} C_VEL
LIN {X 0,Y 343.118,Z 915.512,A -85,B 0,C 180,E1 25534.339,E2 25534.339} C_VEL
LIN {X 0,Y 347.913,Z 906.391,A -85,B 0,C 180,E1 25535.063,E2 25535.063} C_VEL
LIN {X 0,Y 346.865,Z 889.156,A -85,B 0,C 180,E1 25540.214,E2 25540.214} C_VEL
LIN {X 0,Y 344.728,Z 875.259,A -85,B 0,C 180,E1 25545.884,E2 25545.884} C_VEL
LIN {X 0,Y 342.883,Z 864.906,A -85,B 0,C 180,E1 25552.386,E2 25552.386} C_VEL
LIN {X 0,Y 342.306,Z 860.924,A -85,B 0,C 180,E1 25557.467,E2 25557.467} C_VEL
LIN {X 0,Y 342.312,Z 860.373,A -85,B 0,C 180,E1 25560.005,E2 25560.005} C_VEL
LIN {X 0,Y 342.366,Z 866.787,A -85,B 0,C 180,E1 25567.635,E2 25567.635} C_VEL
LIN {X 0,Y 343.658,Z 877.833,A -85,B 0,C 180,E1 25574.048,E2 25574.048} C_VEL
LIN {X 0,Y 344.708,Z 892.298,A -85,B 0,C 180,E1 25579.59,E2 25579.59} C_VEL
LIN {X 0,Y 344.735,Z 907,A -85,B 0,C 180,E1 25583.997,E2 25583.997} C_VEL
LIN {X 0,Y 321.678,Z 945.34,A -85,B 0,C 180,E1 25588.11,E2 25588.11} C_VEL
LIN {X 0,Y 307.317,Z 965.526,A -85,B 0,C 180,E1 25591.036,E2 25591.036} C_VEL
LIN {X 0,Y 296.325,Z 977.124,A -85,B 0,C 180,E1 25592.428,E2 25592.428} C_VEL
LIN {X 0,Y 285.158,Z 988.052,A -85,B 0,C 180,E1 25593.994,E2 25593.994} C_VEL
LIN {X 0,Y 261.829,Z 1014.038,A -85,B 0,C 180,E1 25601.203,E2 25601.203} C_VEL
LIN {X 0,Y 241.965,Z 1034.473,A -85,B 0,C 180,E1 25610.065,E2 25610.065} C_VEL
LIN {X 0,Y 227.558,Z 1049.552,A -85,B 0,C 180,E1 25620.711,E2 25620.711} C_VEL
LIN {X 0,Y 219.822,Z 1058.517,A -85,B 0,C 180,E1 25631.929,E2 25631.929} C_VEL
LIN {X 0,Y 217.145,Z 1062.273,A -85,B 0,C 180,E1 25641.979,E2 25641.979} C_VEL
LIN {X 0,Y 217.436,Z 1062.446,A -85,B 0,C 180,E1 25650.002,E2 25650.002} C_VEL
LIN {X 0,Y 217.972,Z 1060.286,A -85,B 0,C 180,E1 25657.994,E2 25657.994} C_VEL
LIN {X 0,Y 221.671,Z 1054.189,A -85,B 0,C 180,E1 25667.918,E2 25667.918} C_VEL
LIN {X 0,Y 231.819,Z 1041.432,A -85,B 0,C 180,E1 25679.361,E2 25679.361} C_VEL
LIN {X 0,Y 247.196,Z 1024.054,A -85,B 0,C 180,E1 25688.931,E2 25688.931} C_VEL
LIN {X 0,Y 268.057,Z 1000.221,A -85,B 0,C 180,E1 25697.303,E2 25697.303} C_VEL
LIN {X 0,Y 292.196,Z 969.854,A -85,B 0,C 180,E1 25704.132,E2 25704.132} C_VEL
LIN {X 0,Y 316.901,Z 933.606,A -85,B 0,C 180,E1 25709.403,E2 25709.403} C_VEL
LIN {X 0,Y 333.073,Z 905.431,A -85,B 0,C 180,E1 25712.265,E2 25712.265} C_VEL
LIN {X 0,Y 333.149,Z 887.287,A -85,B 0,C 180,E1 25717.439,E2 25717.439} C_VEL
LIN {X 0,Y 331.656,Z 871.012,A -85,B 0,C 180,E1 25723.648,E2 25723.648} C_VEL
LIN {X 0,Y 330.205,Z 860.805,A -85,B 0,C 180,E1 25729.417,E2 25729.417} C_VEL
LIN {X 0,Y 329.616,Z 855.411,A -85,B 0,C 180,E1 25734.72,E2 25734.72} C_VEL
LIN {X 0,Y 329.965,Z 853.514,A -85,B 0,C 180,E1 25737.363,E2 25737.363} C_VEL
LIN {X 0,Y 330.119,Z 853.393,A -85,B 0,C 180,E1 25739.995,E2 25739.995} C_VEL
LIN {X 0,Y 330.862,Z 858.709,A -85,B 0,C 180,E1 25746.57,E2 25746.57} C_VEL
LIN {X 0,Y 333.024,Z 869.874,A -85,B 0,C 180,E1 25753.146,E2 25753.146} C_VEL
LIN {X 0,Y 335.434,Z 885.881,A -85,B 0,C 180,E1 25759.286,E2 25759.286} C_VEL
LIN {X 0,Y 336.297,Z 904.243,A -85,B 0,C 180,E1 25764.436,E2 25764.436} C_VEL
LIN {X 0,Y 313.904,Z 943.85,A -85,B 0,C 180,E1 25768.23,E2 25768.23} C_VEL
LIN {X 0,Y 290.02,Z 978.821,A -85,B 0,C 180,E1 25773.275,E2 25773.275} C_VEL
LIN {X 0,Y 265.593,Z 1010.051,A -85,B 0,C 180,E1 25780.256,E2 25780.256} C_VEL
LIN {X 0,Y 243.897,Z 1035.6,A -85,B 0,C 180,E1 25789.276,E2 25789.276} C_VEL
LIN {X 0,Y 227.46,Z 1055.404,A -85,B 0,C 180,E1 25800.688,E2 25800.688} C_VEL
LIN {X 0,Y 219.666,Z 1066.92,A -85,B 0,C 180,E1 25811.912,E2 25811.912} C_VEL
LIN {X 0,Y 217.278,Z 1072.654,A -85,B 0,C 180,E1 25821.98,E2 25821.98} C_VEL
LIN {X 0,Y 217.464,Z 1074.228,A -85,B 0,C 180,E1 25829.998,E2 25829.998} C_VEL
LIN {X 0,Y 217.254,Z 1073.237,A -85,B 0,C 180,E1 25838.017,E2 25838.017} C_VEL
LIN {X 0,Y 219.697,Z 1068.491,A -85,B 0,C 180,E1 25848.081,E2 25848.081} C_VEL
LIN {X 0,Y 227.821,Z 1057.897,A -85,B 0,C 180,E1 25859.388,E2 25859.388} C_VEL
LIN {X 0,Y 242.664,Z 1041.589,A -85,B 0,C 180,E1 25869.797,E2 25869.797} C_VEL
LIN {X 0,Y 263.912,Z 1018.694,A -85,B 0,C 180,E1 25878.861,E2 25878.861} C_VEL
LIN {X 0,Y 289.499,Z 988.961,A -85,B 0,C 180,E1 25886.197,E2 25886.197} C_VEL
LIN {X 0,Y 315.423,Z 954.378,A -85,B 0,C 180,E1 25891.615,E2 25891.615} C_VEL
LIN {X 0,Y 339.598,Z 915.741,A -85,B 0,C 180,E1 25895.535,E2 25895.535} C_VEL
LIN {X 0,Y 342.763,Z 909.07,A -85,B 0,C 180,E1 25896.213,E2 25896.213} C_VEL
LIN {X 0,Y 341.852,Z 891.445,A -85,B 0,C 180,E1 25901.928,E2 25901.928} C_VEL
LIN {X 0,Y 340.091,Z 878.411,A -85,B 0,C 180,E1 25907.953,E2 25907.953} C_VEL
LIN {X 0,Y 338.984,Z 870.895,A -85,B 0,C 180,E1 25913.588,E2 25913.588} C_VEL
LIN {X 0,Y 338.764,Z 868.05,A -85,B 0,C 180,E1 25917.441,E2 25917.441} C_VEL
LIN {X 0,Y 338.765,Z 867.503,A -85,B 0,C 180,E1 25920.005,E2 25920.005} C_VEL
LIN {X 0,Y 338.495,Z 873.929,A -85,B 0,C 180,E1 25927.723,E2 25927.723} C_VEL
LIN {X 0,Y 339.362,Z 883.851,A -85,B 0,C 180,E1 25933.567,E2 25933.567} C_VEL
LIN {X 0,Y 339.875,Z 898.365,A -85,B 0,C 180,E1 25939.284,E2 25939.284} C_VEL
LIN {X 0,Y 339.373,Z 911.133,A -85,B 0,C 180,E1 25943.193,E2 25943.193} C_VEL
LIN {X 0,Y 315.965,Z 948.289,A -85,B 0,C 180,E1 25947.195,E2 25947.195} C_VEL
LIN {X 0,Y 290.379,Z 981.972,A -85,B 0,C 180,E1 25952.702,E2 25952.702} C_VEL
LIN {X 0,Y 285.158,Z 988.052,A -85,B 0,C 180,E1 25953.994,E2 25953.994} C_VEL
LIN {X 0,Y 273.819,Z 998.355,A -85,B 0,C 180,E1 25955.763,E2 25955.763} C_VEL
LIN {X 0,Y 262.526,Z 1007.935,A -85,B 0,C 180,E1 25957.764,E2 25957.764} C_VEL
LIN {X 0,Y 240.914,Z 1029.664,A -85,B 0,C 180,E1 25966.22,E2 25966.22} C_VEL
LIN {X 0,Y 224.498,Z 1045.665,A -85,B 0,C 180,E1 25976.161,E2 25976.161} C_VEL
LIN {X 0,Y 214.704,Z 1055.743,A -85,B 0,C 180,E1 25986.587,E2 25986.587} C_VEL
LIN {X 0,Y 210.027,Z 1061.477,A -85,B 0,C 180,E1 25997.501,E2 25997.501} C_VEL
LIN {X 0,Y 209.552,Z 1062.66,A -85,B 0,C 180,E1 26010.002,E2 26010.002} C_VEL
LIN {X 0,Y 210.112,Z 1060.515,A -85,B 0,C 180,E1 26018.296,E2 26018.296} C_VEL
LIN {X 0,Y 214.071,Z 1054.433,A -85,B 0,C 180,E1 26028.577,E2 26028.577} C_VEL
LIN {X 0,Y 224.856,Z 1041.699,A -85,B 0,C 180,E1 26040.364,E2 26040.364} C_VEL
LIN {X 0,Y 240.811,Z 1024.569,A -85,B 0,C 180,E1 26050.032,E2 26050.032} C_VEL
LIN {X 0,Y 262.681,Z 1000.541,A -85,B 0,C 180,E1 26058.59,E2 26058.59} C_VEL
LIN {X 0,Y 287.587,Z 970.205,A -85,B 0,C 180,E1 26065.423,E2 26065.423} C_VEL
LIN {X 0,Y 312.925,Z 933.998,A -85,B 0,C 180,E1 26070.657,E2 26070.657} C_VEL
LIN {X 0,Y 328.103,Z 908.136,A -85,B 0,C 180,E1 26073.351,E2 26073.351} C_VEL
LIN {X 0,Y 328.249,Z 889.199,A -85,B 0,C 180,E1 26079.206,E2 26079.206} C_VEL
LIN {X 0,Y 327.206,Z 874.905,A -85,B 0,C 180,E1 26085.238,E2 26085.238} C_VEL
LIN {X 0,Y 326.29,Z 864.737,A -85,B 0,C 180,E1 26091.986,E2 26091.986} C_VEL
LIN {X 0,Y 326.426,Z 860.67,A -85,B 0,C 180,E1 26097.334,E2 26097.334} C_VEL
LIN {X 0,Y 326.618,Z 860.52,A -85,B 0,C 180,E1 26099.995,E2 26099.995} C_VEL
LIN {X 0,Y 327.251,Z 866.013,A -85,B 0,C 180,E1 26106.643,E2 26106.643} C_VEL
LIN {X 0,Y 329.039,Z 877.395,A -85,B 0,C 180,E1 26113.308,E2 26113.308} C_VEL
LIN {X 0,Y 330.766,Z 892.251,A -85,B 0,C 180,E1 26119.047,E2 26119.047} C_VEL
LIN {X 0,Y 331.261,Z 906.625,A -85,B 0,C 180,E1 26123.291,E2 26123.291} C_VEL
LIN {X 0,Y 309.442,Z 944.546,A -85,B 0,C 180,E1 26127.039,E2 26127.039} C_VEL
LIN {X 0,Y 284.436,Z 980.019,A -85,B 0,C 180,E1 26132.186,E2 26132.186} C_VEL
LIN {X 0,Y 259.279,Z 1011.005,A -85,B 0,C 180,E1 26139.245,E2 26139.245} C_VEL
LIN {X 0,Y 237.747,Z 1035.311,A -85,B 0,C 180,E1 26147.987,E2 26147.987} C_VEL
LIN {X 0,Y 220.357,Z 1055.196,A -85,B 0,C 180,E1 26159.694,E2 26159.694} C_VEL
LIN {X 0,Y 212.019,Z 1066.677,A -85,B 0,C 180,E1 26171.236,E2 26171.236} C_VEL
LIN {X 0,Y 209.393,Z 1072.427,A -85,B 0,C 180,E1 26181.676,E2 26181.676} C_VEL
LIN {X 0,Y 209.573,Z 1074.014,A -85,B 0,C 180,E1 26189.998,E2 26189.998} C_VEL
LIN {X 0,Y 209.368,Z 1073.034,A -85,B 0,C 180,E1 26198.321,E2 26198.321} C_VEL
LIN {X 0,Y 212.059,Z 1068.298,A -85,B 0,C 180,E1 26208.756,E2 26208.756} C_VEL
LIN {X 0,Y 220.598,Z 1057.886,A -85,B 0,C 180,E1 26220.289,E2 26220.289} C_VEL
LIN {X 0,Y 236.443,Z 1041.433,A -85,B 0,C 180,E1 26231.065,E2 26231.065} C_VEL
LIN {X 0,Y 258.7,Z 1018.479,A -85,B 0,C 180,E1 26240.246,E2 26240.246} C_VEL
LIN {X 0,Y 285.049,Z 988.86,A -85,B 0,C 180,E1 26247.558,E2 26247.558} C_VEL
LIN {X 0,Y 311.684,Z 954.314,A -85,B 0,C 180,E1 26252.914,E2 26252.914} C_VEL
LIN {X 0,Y 336.361,Z 915.719,A -85,B 0,C 180,E1 26256.776,E2 26256.776} C_VEL
LIN {X 0,Y 337.606,Z 912.18,A -85,B 0,C 180,E1 26257.329,E2 26257.329} C_VEL
LIN {X 0,Y 337.149,Z 896.269,A -85,B 0,C 180,E1 26262.771,E2 26262.771} C_VEL
LIN {X 0,Y 335.94,Z 884.292,A -85,B 0,C 180,E1 26268.632,E2 26268.632} C_VEL
LIN {X 0,Y 334.985,Z 877.195,A -85,B 0,C 180,E1 26274.389,E2 26274.389} C_VEL
LIN {X 0,Y 334.977,Z 874.484,A -85,B 0,C 180,E1 26280.005,E2 26280.005} C_VEL
LIN {X 0,Y 334.503,Z 879.428,A -85,B 0,C 180,E1 26286.508,E2 26286.508} C_VEL
LIN {X 0,Y 334.883,Z 888.446,A -85,B 0,C 180,E1 26292.417,E2 26292.417} C_VEL
LIN {X 0,Y 335.008,Z 902.154,A -85,B 0,C 180,E1 26298.212,E2 26298.212} C_VEL
LIN {X 0,Y 334.399,Z 913.567,A -85,B 0,C 180,E1 26301.959,E2 26301.959} C_VEL
LIN {X 0,Y 329.966,Z 921.781,A -85,B 0,C 180,E1 26302.889,E2 26302.889} C_VEL
LIN {X 0,Y 304.76,Z 958.638,A -85,B 0,C 180,E1 26307.277,E2 26307.277} C_VEL
LIN {X 0,Y 277.417,Z 991.952,A -85,B 0,C 180,E1 26313.456,E2 26313.456} C_VEL
LIN {X 0,Y 262.526,Z 1007.935,A -85,B 0,C 180,E1 26317.764,E2 26317.764} C_VEL
LIN {X 0,Y 251.202,Z 1016.855,A -85,B 0,C 180,E1 26320.014,E2 26320.014} C_VEL
LIN {X 0,Y 240.228,Z 1025.005,A -85,B 0,C 180,E1 26322.568,E2 26322.568} C_VEL
LIN {X 0,Y 220.46,Z 1043.32,A -85,B 0,C 180,E1 26333.028,E2 26333.028} C_VEL
LIN {X 0,Y 208.436,Z 1054.798,A -85,B 0,C 180,E1 26344.139,E2 26344.139} C_VEL
LIN {X 0,Y 202.224,Z 1061.677,A -85,B 0,C 180,E1 26357.01,E2 26357.01} C_VEL
LIN {X 0,Y 201.639,Z 1062.875,A -85,B 0,C 180,E1 26370.002,E2 26370.002} C_VEL
LIN {X 0,Y 202.257,Z 1060.744,A -85,B 0,C 180,E1 26378.62,E2 26378.62} C_VEL
LIN {X 0,Y 206.525,Z 1054.677,A -85,B 0,C 180,E1 26389.282,E2 26389.282} C_VEL
LIN {X 0,Y 217.985,Z 1041.965,A -85,B 0,C 180,E1 26401.427,E2 26401.427} C_VEL
LIN {X 0,Y 235.972,Z 1023.528,A -85,B 0,C 180,E1 26411.881,E2 26411.881} C_VEL
LIN {X 0,Y 258.575,Z 999.553,A -85,B 0,C 180,E1 26420.284,E2 26420.284} C_VEL
LIN {X 0,Y 283.123,Z 970.554,A -85,B 0,C 180,E1 26426.756,E2 26426.756} C_VEL
LIN {X 0,Y 309.1,Z 934.39,A -85,B 0,C 180,E1 26431.944,E2 26431.944} C_VEL
LIN {X 0,Y 322.776,Z 911.961,A -85,B 0,C 180,E1 26434.23,E2 26434.23} C_VEL
LIN {X 0,Y 323.598,Z 895.492,A -85,B 0,C 180,E1 26439.49,E2 26439.49} C_VEL
LIN {X 0,Y 323.068,Z 881.057,A -85,B 0,C 180,E1 26445.739,E2 26445.739} C_VEL
LIN {X 0,Y 322.527,Z 871.931,A -85,B 0,C 180,E1 26451.892,E2 26451.892} C_VEL
LIN {X 0,Y 322.869,Z 867.824,A -85,B 0,C 180,E1 26457.305,E2 26457.305} C_VEL
LIN {X 0,Y 323.07,Z 867.648,A -85,B 0,C 180,E1 26459.995,E2 26459.995} C_VEL
LIN {X 0,Y 323.513,Z 873.238,A -85,B 0,C 180,E1 26466.72,E2 26466.72} C_VEL
LIN {X 0,Y 324.802,Z 883.419,A -85,B 0,C 180,E1 26472.798,E2 26472.798} C_VEL
LIN {X 0,Y 326.003,Z 898.111,A -85,B 0,C 180,E1 26478.632,E2 26478.632} C_VEL
LIN {X 0,Y 325.994,Z 910.642,A -85,B 0,C 180,E1 26482.444,E2 26482.444} C_VEL
LIN {X 0,Y 303.679,Z 947.372,A -85,B 0,C 180,E1 26486.071,E2 26486.071} C_VEL
LIN {X 0,Y 279.329,Z 980.737,A -85,B 0,C 180,E1 26490.973,E2 26490.973} C_VEL
LIN {X 0,Y 254.182,Z 1010.699,A -85,B 0,C 180,E1 26497.817,E2 26497.817} C_VEL
LIN {X 0,Y 231.364,Z 1035.443,A -85,B 0,C 180,E1 26506.823,E2 26506.823} C_VEL
LIN {X 0,Y 213.695,Z 1054.561,A -85,B 0,C 180,E1 26518.302,E2 26518.302} C_VEL
LIN {X 0,Y 204.391,Z 1066.434,A -85,B 0,C 180,E1 26530.508,E2 26530.508} C_VEL
LIN {X 0,Y 201.507,Z 1072.199,A -85,B 0,C 180,E1 26541.347,E2 26541.347} C_VEL
LIN {X 0,Y 201.662,Z 1073.8,A -85,B 0,C 180,E1 26549.998,E2 26549.998} C_VEL
LIN {X 0,Y 201.482,Z 1072.83,A -85,B 0,C 180,E1 26558.65,E2 26558.65} C_VEL
LIN {X 0,Y 204.438,Z 1068.104,A -85,B 0,C 180,E1 26569.483,E2 26569.483} C_VEL
LIN {X 0,Y 214.138,Z 1057.133,A -85,B 0,C 180,E1 26581.89,E2 26581.89} C_VEL
LIN {X 0,Y 230.334,Z 1041.277,A -85,B 0,C 180,E1 26592.402,E2 26592.402} C_VEL
LIN {X 0,Y 253.593,Z 1018.349,A -85,B 0,C 180,E1 26601.655,E2 26601.655} C_VEL
LIN {X 0,Y 280.784,Z 988.759,A -85,B 0,C 180,E1 26608.954,E2 26608.954} C_VEL
LIN {X 0,Y 308.096,Z 954.251,A -85,B 0,C 180,E1 26614.249,E2 26614.249} C_VEL
LIN {X 0,Y 332.235,Z 917.403,A -85,B 0,C 180,E1 26617.903,E2 26617.903} C_VEL
LIN {X 0,Y 332.531,Z 903.17,A -85,B 0,C 180,E1 26622.776,E2 26622.776} C_VEL
LIN {X 0,Y 331.666,Z 890.899,A -85,B 0,C 180,E1 26628.808,E2 26628.808} C_VEL
LIN {X 0,Y 331.075,Z 883.859,A -85,B 0,C 180,E1 26634.752,E2 26634.752} C_VEL
LIN {X 0,Y 331.121,Z 881.431,A -85,B 0,C 180,E1 26640.005,E2 26640.005} C_VEL
LIN {X 0,Y 330.413,Z 886.443,A -85,B 0,C 180,E1 26646.589,E2 26646.589} C_VEL
LIN {X 0,Y 330.525,Z 895.694,A -85,B 0,C 180,E1 26652.583,E2 26652.583} C_VEL
LIN {X 0,Y 330.005,Z 909.849,A -85,B 0,C 180,E1 26658.498,E2 26658.498} C_VEL
LIN {X 0,Y 329.286,Z 917.381,A -85,B 0,C 180,E1 26661.059,E2 26661.059} C_VEL
LIN {X 0,Y 306.274,Z 951.87,A -85,B 0,C 180,E1 26664.979,E2 26664.979} C_VEL
LIN {X 0,Y 280.603,Z 983.627,A -85,B 0,C 180,E1 26670.225,E2 26670.225} C_VEL
LIN {X 0,Y 255.409,Z 1010.336,A -85,B 0,C 180,E1 26677.02,E2 26677.02} C_VEL
LIN {X 0,Y 240.228,Z 1025.005,A -85,B 0,C 180,E1 26682.568,E2 26682.568} C_VEL
LIN {X 0,Y 229.44,Z 1032.443,A -85,B 0,C 180,E1 26685.416,E2 26685.416} C_VEL
LIN {X 0,Y 218.96,Z 1039.13,A -85,B 0,C 180,E1 26688.586,E2 26688.586} C_VEL
LIN {X 0,Y 202.993,Z 1053.285,A -85,B 0,C 180,E1 26700.974,E2 26700.974} C_VEL
LIN {X 0,Y 195.968,Z 1060.212,A -85,B 0,C 180,E1 26711.984,E2 26711.984} C_VEL
LIN {X 0,Y 193.524,Z 1062.88,A -85,B 0,C 180,E1 26720.992,E2 26720.992} C_VEL
LIN {X 0,Y 193.737,Z 1063.089,A -85,B 0,C 180,E1 26730.002,E2 26730.002} C_VEL
LIN {X 0,Y 194.411,Z 1060.972,A -85,B 0,C 180,E1 26738.971,E2 26738.971} C_VEL
LIN {X 0,Y 199.007,Z 1054.921,A -85,B 0,C 180,E1 26750.042,E2 26750.042} C_VEL
LIN {X 0,Y 211.182,Z 1042.232,A -85,B 0,C 180,E1 26762.562,E2 26762.562} C_VEL
LIN {X 0,Y 229.466,Z 1024.403,A -85,B 0,C 180,E1 26772.96,E2 26772.96} C_VEL
LIN {X 0,Y 253.528,Z 999.871,A -85,B 0,C 180,E1 26781.678,E2 26781.678} C_VEL
LIN {X 0,Y 278.814,Z 970.902,A -85,B 0,C 180,E1 26788.132,E2 26788.132} C_VEL
LIN {X 0,Y 305.436,Z 934.78,A -85,B 0,C 180,E1 26793.263,E2 26793.263} C_VEL
LIN {X 0,Y 317.742,Z 914.711,A -85,B 0,C 180,E1 26795.41,E2 26795.41} C_VEL
LIN {X 0,Y 318.75,Z 899.586,A -85,B 0,C 180,E1 26800.557,E2 26800.557} C_VEL
LIN {X 0,Y 318.728,Z 887.082,A -85,B 0,C 180,E1 26806.243,E2 26806.243} C_VEL
LIN {X 0,Y 318.613,Z 879.045,A -85,B 0,C 180,E1 26811.792,E2 26811.792} C_VEL
LIN {X 0,Y 319.042,Z 874.835,A -85,B 0,C 180,E1 26817.273,E2 26817.273} C_VEL
LIN {X 0,Y 319.278,Z 874.649,A -85,B 0,C 180,E1 26819.995,E2 26819.995} C_VEL
LIN {X 0,Y 319.584,Z 880.357,A -85,B 0,C 180,E1 26826.803,E2 26826.803} C_VEL
LIN {X 0,Y 320.495,Z 890.841,A -85,B 0,C 180,E1 26832.974,E2 26832.974} C_VEL
LIN {X 0,Y 321.119,Z 905.504,A -85,B 0,C 180,E1 26838.763,E2 26838.763} C_VEL
LIN {X 0,Y 320.484,Z 914.778,A -85,B 0,C 180,E1 26841.475,E2 26841.475} C_VEL
LIN {X 0,Y 294.567,Z 955.165,A -85,B 0,C 180,E1 26845.672,E2 26845.672} C_VEL
LIN {X 0,Y 268.331,Z 988.762,A -85,B 0,C 180,E1 26851.105,E2 26851.105} C_VEL
LIN {X 0,Y 241.514,Z 1018.61,A -85,B 0,C 180,E1 26858.854,E2 26858.854} C_VEL
LIN {X 0,Y 218.771,Z 1041.885,A -85,B 0,C 180,E1 26868.843,E2 26868.843} C_VEL
LIN {X 0,Y 202.778,Z 1058.626,A -85,B 0,C 180,E1 26880.936,E2 26880.936} C_VEL
LIN {X 0,Y 195.052,Z 1068.964,A -85,B 0,C 180,E1 26894.219,E2 26894.219} C_VEL
LIN {X 0,Y 193.38,Z 1073.093,A -85,B 0,C 180,E1 26905.503,E2 26905.503} C_VEL
LIN {X 0,Y 193.778,Z 1073.587,A -85,B 0,C 180,E1 26909.998,E2 26909.998} C_VEL
LIN {X 0,Y 193.601,Z 1072.626,A -85,B 0,C 180,E1 26919.004,E2 26919.004} C_VEL
LIN {X 0,Y 196.83,Z 1067.909,A -85,B 0,C 180,E1 26930.268,E2 26930.268} C_VEL
LIN {X 0,Y 207.242,Z 1056.956,A -85,B 0,C 180,E1 26943.084,E2 26943.084} C_VEL
LIN {X 0,Y 224.256,Z 1041.226,A -85,B 0,C 180,E1 26953.758,E2 26953.758} C_VEL
LIN {X 0,Y 248.643,Z 1018.219,A -85,B 0,C 180,E1 26963.12,E2 26963.12} C_VEL
LIN {X 0,Y 276.689,Z 988.676,A -85,B 0,C 180,E1 26970.384,E2 26970.384} C_VEL
LIN {X 0,Y 304.682,Z 954.188,A -85,B 0,C 180,E1 26975.614,E2 26975.614} C_VEL
LIN {X 0,Y 326.918,Z 921.229,A -85,B 0,C 180,E1 26978.874,E2 26978.874} C_VEL
LIN {X 0,Y 327.685,Z 908.454,A -85,B 0,C 180,E1 26983.395,E2 26983.395} C_VEL
LIN {X 0,Y 327.316,Z 896.911,A -85,B 0,C 180,E1 26989.333,E2 26989.333} C_VEL
LIN {X 0,Y 326.93,Z 890.69,A -85,B 0,C 180,E1 26994.686,E2 26994.686} C_VEL
LIN {X 0,Y 327.047,Z 888.277,A -85,B 0,C 180,E1 27000.005,E2 27000.005} C_VEL
LIN {X 0,Y 326.174,Z 893.371,A -85,B 0,C 180,E1 27006.675,E2 27006.675} C_VEL
LIN {X 0,Y 325.832,Z 902.69,A -85,B 0,C 180,E1 27012.7,E2 27012.7} C_VEL
LIN {X 0,Y 324.793,Z 916.131,A -85,B 0,C 180,E1 27018.362,E2 27018.362} C_VEL
LIN {X 0,Y 324.217,Z 921.298,A -85,B 0,C 180,E1 27020.15,E2 27020.15} C_VEL
LIN {X 0,Y 297.687,Z 958.768,A -85,B 0,C 180,E1 27024.506,E2 27024.506} C_VEL
LIN {X 0,Y 269.335,Z 991.569,A -85,B 0,C 180,E1 27030.429,E2 27030.429} C_VEL
LIN {X 0,Y 242.66,Z 1017.978,A -85,B 0,C 180,E1 27038.177,E2 27038.177} C_VEL
LIN {X 0,Y 218.96,Z 1039.13,A -85,B 0,C 180,E1 27048.586,E2 27048.586} C_VEL
LIN {X 0,Y 209.138,Z 1045.081,A -85,B 0,C 180,E1 27052.136,E2 27052.136} C_VEL
LIN {X 0,Y 199.841,Z 1050.14,A -85,B 0,C 180,E1 27056.072,E2 27056.072} C_VEL
LIN {X 0,Y 189.424,Z 1059.281,A -85,B 0,C 180,E1 27068.902,E2 27068.902} C_VEL
LIN {X 0,Y 185.659,Z 1063.083,A -85,B 0,C 180,E1 27080.607,E2 27080.607} C_VEL
LIN {X 0,Y 185.823,Z 1063.303,A -85,B 0,C 180,E1 27090.002,E2 27090.002} C_VEL
LIN {X 0,Y 186.571,Z 1061.201,A -85,B 0,C 180,E1 27099.351,E2 27099.351} C_VEL
LIN {X 0,Y 193.091,Z 1053.493,A -85,B 0,C 180,E1 27113.106,E2 27113.106} C_VEL
LIN {X 0,Y 207.408,Z 1039.873,A -85,B 0,C 180,E1 27125.771,E2 27125.771} C_VEL
LIN {X 0,Y 230.297,Z 1018.452,A -85,B 0,C 180,E1 27137.061,E2 27137.061} C_VEL
LIN {X 0,Y 256.115,Z 992.343,A -85,B 0,C 180,E1 27145.184,E2 27145.184} C_VEL
LIN {X 0,Y 284.453,Z 959.082,A -85,B 0,C 180,E1 27151.522,E2 27151.522} C_VEL
LIN {X 0,Y 310.959,Z 921.405,A -85,B 0,C 180,E1 27156.028,E2 27156.028} C_VEL
LIN {X 0,Y 312.7,Z 917.741,A -85,B 0,C 180,E1 27156.591,E2 27156.591} C_VEL
LIN {X 0,Y 313.978,Z 903.819,A -85,B 0,C 180,E1 27161.612,E2 27161.612} C_VEL
LIN {X 0,Y 314.346,Z 891.716,A -85,B 0,C 180,E1 27167.601,E2 27167.601} C_VEL
LIN {X 0,Y 314.611,Z 884.761,A -85,B 0,C 180,E1 27173.079,E2 27173.079} C_VEL
LIN {X 0,Y 315.181,Z 881.789,A -85,B 0,C 180,E1 27177.239,E2 27177.239} C_VEL
LIN {X 0,Y 315.411,Z 881.606,A -85,B 0,C 180,E1 27179.995,E2 27179.995} C_VEL
LIN {X 0,Y 315.538,Z 887.435,A -85,B 0,C 180,E1 27186.891,E2 27186.891} C_VEL
LIN {X 0,Y 316.095,Z 898.167,A -85,B 0,C 180,E1 27193.158,E2 27193.158} C_VEL
LIN {X 0,Y 316.092,Z 911.783,A -85,B 0,C 180,E1 27198.544,E2 27198.544} C_VEL
LIN {X 0,Y 315.4,Z 918.07,A -85,B 0,C 180,E1 27200.434,E2 27200.434} C_VEL
LIN {X 0,Y 291.149,Z 954.784,A -85,B 0,C 180,E1 27204.226,E2 27204.226} C_VEL
LIN {X 0,Y 263.977,Z 988.705,A -85,B 0,C 180,E1 27209.644,E2 27209.644} C_VEL
LIN {X 0,Y 236.469,Z 1018.304,A -85,B 0,C 180,E1 27217.31,E2 27217.31} C_VEL
LIN {X 0,Y 212.664,Z 1041.608,A -85,B 0,C 180,E1 27227.392,E2 27227.392} C_VEL
LIN {X 0,Y 195.691,Z 1058.367,A -85,B 0,C 180,E1 27239.776,E2 27239.776} C_VEL
LIN {X 0,Y 187.33,Z 1068.728,A -85,B 0,C 180,E1 27253.551,E2 27253.551} C_VEL
LIN {X 0,Y 185.467,Z 1072.872,A -85,B 0,C 180,E1 27265.311,E2 27265.311} C_VEL
LIN {X 0,Y 185.865,Z 1073.373,A -85,B 0,C 180,E1 27269.998,E2 27269.998} C_VEL
LIN {X 0,Y 186.243,Z 1071.611,A -85,B 0,C 180,E1 27282.515,E2 27282.515} C_VEL
LIN {X 0,Y 192.699,Z 1064.142,A -85,B 0,C 180,E1 27296.459,E2 27296.459} C_VEL
LIN {X 0,Y 207.945,Z 1050.195,A -85,B 0,C 180,E1 27309.615,E2 27309.615} C_VEL
LIN {X 0,Y 228.761,Z 1031.838,A -85,B 0,C 180,E1 27319.621,E2 27319.621} C_VEL
LIN {X 0,Y 254.155,Z 1007.984,A -85,B 0,C 180,E1 27327.554,E2 27327.554} C_VEL
LIN {X 0,Y 282.807,Z 977.221,A -85,B 0,C 180,E1 27333.833,E2 27333.833} C_VEL
LIN {X 0,Y 310.65,Z 941.503,A -85,B 0,C 180,E1 27338.393,E2 27338.393} C_VEL
LIN {X 0,Y 321.816,Z 924.859,A -85,B 0,C 180,E1 27339.896,E2 27339.896} C_VEL
LIN {X 0,Y 322.898,Z 912.991,A -85,B 0,C 180,E1 27344.35,E2 27344.35} C_VEL
LIN {X 0,Y 322.82,Z 902.224,A -85,B 0,C 180,E1 27350.322,E2 27350.322} C_VEL
LIN {X 0,Y 322.742,Z 897.519,A -85,B 0,C 180,E1 27354.617,E2 27354.617} C_VEL
LIN {X 0,Y 322.876,Z 895.049,A -85,B 0,C 180,E1 27360.005,E2 27360.005} C_VEL
LIN {X 0,Y 321.789,Z 900.218,A -85,B 0,C 180,E1 27366.766,E2 27366.766} C_VEL
LIN {X 0,Y 321.126,Z 909.283,A -85,B 0,C 180,E1 27372.614,E2 27372.614} C_VEL
LIN {X 0,Y 319.485,Z 923.04,A -85,B 0,C 180,E1 27378.445,E2 27378.445} C_VEL
LIN {X 0,Y 318.587,Z 925.931,A -85,B 0,C 180,E1 27379.297,E2 27379.297} C_VEL
LIN {X 0,Y 292.924,Z 960.698,A -85,B 0,C 180,E1 27383.329,E2 27383.329} C_VEL
LIN {X 0,Y 263.538,Z 993.466,A -85,B 0,C 180,E1 27389.324,E2 27389.324} C_VEL
LIN {X 0,Y 236.362,Z 1019.343,A -85,B 0,C 180,E1 27397.081,E2 27397.081} C_VEL
LIN {X 0,Y 211.971,Z 1040.053,A -85,B 0,C 180,E1 27407.639,E2 27407.639} C_VEL
LIN {X 0,Y 199.841,Z 1050.14,A -85,B 0,C 180,E1 27416.072,E2 27416.072} C_VEL
LIN {X 0,Y 191.302,Z 1054.526,A -85,B 0,C 180,E1 27420.381,E2 27420.381} C_VEL
LIN {X 0,Y 183.626,Z 1058.029,A -85,B 0,C 180,E1 27425.09,E2 27425.09} C_VEL
LIN {X 0,Y 178.911,Z 1062.27,A -85,B 0,C 180,E1 27435.282,E2 27435.282} C_VEL
LIN {X 0,Y 177.907,Z 1063.518,A -85,B 0,C 180,E1 27450.002,E2 27450.002} C_VEL
LIN {X 0,Y 178.739,Z 1061.43,A -85,B 0,C 180,E1 27459.765,E2 27459.765} C_VEL
LIN {X 0,Y 185.753,Z 1053.745,A -85,B 0,C 180,E1 27474.076,E2 27474.076} C_VEL
LIN {X 0,Y 200.935,Z 1040.144,A -85,B 0,C 180,E1 27487.112,E2 27487.112} C_VEL
LIN {X 0,Y 224.904,Z 1018.751,A -85,B 0,C 180,E1 27498.558,E2 27498.558} C_VEL
LIN {X 0,Y 251.597,Z 992.665,A -85,B 0,C 180,E1 27506.692,E2 27506.692} C_VEL
LIN {X 0,Y 280.537,Z 959.712,A -85,B 0,C 180,E1 27512.913,E2 27512.913} C_VEL
LIN {X 0,Y 306.984,Z 923.135,A -85,B 0,C 180,E1 27517.253,E2 27517.253} C_VEL
LIN {X 0,Y 308.912,Z 912.126,A -85,B 0,C 180,E1 27520.995,E2 27520.995} C_VEL
LIN {X 0,Y 309.864,Z 900.215,A -85,B 0,C 180,E1 27526.563,E2 27526.563} C_VEL
LIN {X 0,Y 310.394,Z 891.651,A -85,B 0,C 180,E1 27532.984,E2 27532.984} C_VEL
LIN {X 0,Y 311.078,Z 888.64,A -85,B 0,C 180,E1 27537.203,E2 27537.203} C_VEL
LIN {X 0,Y 311.357,Z 888.428,A -85,B 0,C 180,E1 27539.995,E2 27539.995} C_VEL
LIN {X 0,Y 311.267,Z 894.411,A -85,B 0,C 180,E1 27546.986,E2 27546.986} C_VEL
LIN {X 0,Y 311.412,Z 905.272,A -85,B 0,C 180,E1 27553.279,E2 27553.279} C_VEL
LIN {X 0,Y 310.791,Z 919.352,A -85,B 0,C 180,E1 27558.793,E2 27558.793} C_VEL
LIN {X 0,Y 309.592,Z 922.606,A -85,B 0,C 180,E1 27559.465,E2 27559.465} C_VEL
LIN {X 0,Y 285.416,Z 957.644,A -85,B 0,C 180,E1 27563.176,E2 27563.176} C_VEL
LIN {X 0,Y 258.493,Z 990.089,A -85,B 0,C 180,E1 27568.431,E2 27568.431} C_VEL
LIN {X 0,Y 230.543,Z 1019.019,A -85,B 0,C 180,E1 27576.042,E2 27576.042} C_VEL
LIN {X 0,Y 206.729,Z 1041.327,A -85,B 0,C 180,E1 27585.86,E2 27585.86} C_VEL
LIN {X 0,Y 188.717,Z 1058.109,A -85,B 0,C 180,E1 27598.534,E2 27598.534} C_VEL
LIN {X 0,Y 179.619,Z 1068.492,A -85,B 0,C 180,E1 27612.823,E2 27612.823} C_VEL
LIN {X 0,Y 177.558,Z 1072.651,A -85,B 0,C 180,E1 27625.102,E2 27625.102} C_VEL
LIN {X 0,Y 177.951,Z 1073.158,A -85,B 0,C 180,E1 27629.998,E2 27629.998} C_VEL
LIN {X 0,Y 177.885,Z 1072.219,A -85,B 0,C 180,E1 27639.808,E2 27639.808} C_VEL
LIN {X 0,Y 181.763,Z 1067.521,A -85,B 0,C 180,E1 27652.033,E2 27652.033} C_VEL
LIN {X 0,Y 193.971,Z 1056.442,A -85,B 0,C 180,E1 27665.867,E2 27665.867} C_VEL
LIN {X 0,Y 213.535,Z 1040.207,A -85,B 0,C 180,E1 27677.178,E2 27677.178} C_VEL
LIN {X 0,Y 240.407,Z 1016.745,A -85,B 0,C 180,E1 27686.635,E2 27686.635} C_VEL
LIN {X 0,Y 269.461,Z 988.034,A -85,B 0,C 180,E1 27693.459,E2 27693.459} C_VEL
LIN {X 0,Y 299.164,Z 953.01,A -85,B 0,C 180,E1 27698.552,E2 27698.552} C_VEL
LIN {X 0,Y 317.183,Z 927.448,A -85,B 0,C 180,E1 27701.192,E2 27701.192} C_VEL
LIN {X 0,Y 318.178,Z 914.394,A -85,B 0,C 180,E1 27706.93,E2 27706.93} C_VEL
LIN {X 0,Y 318.31,Z 905.407,A -85,B 0,C 180,E1 27713.17,E2 27713.17} C_VEL
LIN {X 0,Y 318.509,Z 902.187,A -85,B 0,C 180,E1 27717.585,E2 27717.585} C_VEL
LIN {X 0,Y 318.252,Z 902.176,A -85,B 0,C 180,E1 27720.732,E2 27720.732} C_VEL
LIN {X 0,Y 317.239,Z 906.955,A -85,B 0,C 180,E1 27726.864,E2 27726.864} C_VEL
LIN {X 0,Y 316.208,Z 915.539,A -85,B 0,C 180,E1 27732.459,E2 27732.459} C_VEL
LIN {X 0,Y 314.153,Z 928.198,A -85,B 0,C 180,E1 27737.953,E2 27737.953} C_VEL
LIN {X 0,Y 307.972,Z 937.436,A -85,B 0,C 180,E1 27739.031,E2 27739.031} C_VEL
LIN {X 0,Y 279.683,Z 972.481,A -85,B 0,C 180,E1 27743.636,E2 27743.636} C_VEL
LIN {X 0,Y 249.758,Z 1003.126,A -85,B 0,C 180,E1 27750.165,E2 27750.165} C_VEL
LIN {X 0,Y 222.771,Z 1026.785,A -85,B 0,C 180,E1 27758.532,E2 27758.532} C_VEL
LIN {X 0,Y 199.037,Z 1045.767,A -85,B 0,C 180,E1 27770.37,E2 27770.37} C_VEL
LIN {X 0,Y 184.769,Z 1057.034,A -85,B 0,C 180,E1 27783.452,E2 27783.452} C_VEL
LIN {X 0,Y 183.626,Z 1058.029,A -85,B 0,C 180,E1 27785.09,E2 27785.09} C_VEL
LIN {X 0,Y 176.882,Z 1060.845,A -85,B 0,C 180,E1 27790.131,E2 27790.131} C_VEL
LIN {X 0,Y 170.851,Z 1062.659,A -85,B 0,C 180,E1 27795.552,E2 27795.552} C_VEL
LIN {X 0,Y 169.991,Z 1063.732,A -85,B 0,C 180,E1 27810.002,E2 27810.002} C_VEL
LIN {X 0,Y 172.275,Z 1060.045,A -85,B 0,C 180,E1 27824.591,E2 27824.591} C_VEL
LIN {X 0,Y 182.938,Z 1050.16,A -85,B 0,C 180,E1 27839.806,E2 27839.806} C_VEL
LIN {X 0,Y 201.752,Z 1034.424,A -85,B 0,C 180,E1 27852.535,E2 27852.535} C_VEL
LIN {X 0,Y 227.956,Z 1011.581,A -85,B 0,C 180,E1 27862.917,E2 27862.917} C_VEL
LIN {X 0,Y 257.788,Z 982.026,A -85,B 0,C 180,E1 27870.642,E2 27870.642} C_VEL
LIN {X 0,Y 286.041,Z 948.662,A -85,B 0,C 180,E1 27875.929,E2 27875.929} C_VEL
LIN {X 0,Y 302.086,Z 926.307,A -85,B 0,C 180,E1 27878.359,E2 27878.359} C_VEL
LIN {X 0,Y 304.2,Z 915.003,A -85,B 0,C 180,E1 27882.604,E2 27882.604} C_VEL
LIN {X 0,Y 305.433,Z 903.8,A -85,B 0,C 180,E1 27888.548,E2 27888.548} C_VEL
LIN {X 0,Y 306.322,Z 897.346,A -85,B 0,C 180,E1 27894.317,E2 27894.317} C_VEL
LIN {X 0,Y 306.889,Z 895.442,A -85,B 0,C 180,E1 27897.165,E2 27897.165} C_VEL
LIN {X 0,Y 307.193,Z 895.181,A -85,B 0,C 180,E1 27899.995,E2 27899.995} C_VEL
LIN {X 0,Y 306.994,Z 899.57,A -85,B 0,C 180,E1 27905.661,E2 27905.661} C_VEL
LIN {X 0,Y 306.765,Z 908.174,A -85,B 0,C 180,E1 27911.391,E2 27911.391} C_VEL
LIN {X 0,Y 306.104,Z 919.739,A -85,B 0,C 180,E1 27916.533,E2 27916.533} C_VEL
LIN {X 0,Y 305.228,Z 925.005,A -85,B 0,C 180,E1 27918.28,E2 27918.28} C_VEL
LIN {X 0,Y 279.972,Z 960.226,A -85,B 0,C 180,E1 27922.036,E2 27922.036} C_VEL
LIN {X 0,Y 253.289,Z 991.247,A -85,B 0,C 180,E1 27927.129,E2 27927.129} C_VEL
LIN {X 0,Y 226.054,Z 1018.534,A -85,B 0,C 180,E1 27934.304,E2 27934.304} C_VEL
LIN {X 0,Y 200.938,Z 1041.046,A -85,B 0,C 180,E1 27944.235,E2 27944.235} C_VEL
LIN {X 0,Y 181.415,Z 1058.245,A -85,B 0,C 180,E1 27957.588,E2 27957.588} C_VEL
LIN {X 0,Y 171.932,Z 1068.255,A -85,B 0,C 180,E1 27972.029,E2 27972.029} C_VEL
LIN {X 0,Y 169.646,Z 1072.431,A -85,B 0,C 180,E1 27984.873,E2 27984.873} C_VEL
LIN {X 0,Y 170.035,Z 1072.944,A -85,B 0,C 180,E1 27989.998,E2 27989.998} C_VEL
LIN {X 0,Y 170.234,Z 1071.699,A -85,B 0,C 180,E1 28001.754,E2 28001.754} C_VEL
LIN {X 0,Y 175.851,Z 1065.91,A -85,B 0,C 180,E1 28015.521,E2 28015.521} C_VEL
LIN {X 0,Y 190.536,Z 1053.921,A -85,B 0,C 180,E1 28029.511,E2 28029.511} C_VEL
LIN {X 0,Y 213.927,Z 1035.375,A -85,B 0,C 180,E1 28041.185,E2 28041.185} C_VEL
LIN {X 0,Y 243.014,Z 1010.312,A -85,B 0,C 180,E1 28050.083,E2 28050.083} C_VEL
LIN {X 0,Y 273.01,Z 980.317,A -85,B 0,C 180,E1 28056.326,E2 28056.326} C_VEL
LIN {X 0,Y 301.088,Z 946.625,A -85,B 0,C 180,E1 28060.679,E2 28060.679} C_VEL
LIN {X 0,Y 312.076,Z 931.368,A -85,B 0,C 180,E1 28062.156,E2 28062.156} C_VEL
LIN {X 0,Y 313.321,Z 919.07,A -85,B 0,C 180,E1 28067.951,E2 28067.951} C_VEL
LIN {X 0,Y 313.789,Z 912.1,A -85,B 0,C 180,E1 28073.071,E2 28073.071} C_VEL
LIN {X 0,Y 314.01,Z 908.922,A -85,B 0,C 180,E1 28077.239,E2 28077.239} C_VEL
LIN {X 0,Y 314.048,Z 908.319,A -85,B 0,C 180,E1 28080.005,E2 28080.005} C_VEL
LIN {X 0,Y 312.552,Z 913.64,A -85,B 0,C 180,E1 28086.967,E2 28086.967} C_VEL
LIN {X 0,Y 311.296,Z 921.409,A -85,B 0,C 180,E1 28092.106,E2 28092.106} C_VEL
LIN {X 0,Y 308.911,Z 932.651,A -85,B 0,C 180,E1 28097.123,E2 28097.123} C_VEL
LIN {X 0,Y 282.241,Z 966.103,A -85,B 0,C 180,E1 28101.114,E2 28101.114} C_VEL
LIN {X 0,Y 254.099,Z 995.409,A -85,B 0,C 180,E1 28106.55,E2 28106.55} C_VEL
LIN {X 0,Y 227.444,Z 1019.135,A -85,B 0,C 180,E1 28113.612,E2 28113.612} C_VEL
LIN {X 0,Y 200.764,Z 1039.958,A -85,B 0,C 180,E1 28124.189,E2 28124.189} C_VEL
LIN {X 0,Y 181.764,Z 1054.05,A -85,B 0,C 180,E1 28137.534,E2 28137.534} C_VEL
LIN {X 0,Y 173.152,Z 1060.806,A -85,B 0,C 180,E1 28149.511,E2 28149.511} C_VEL
LIN {X 0,Y 170.851,Z 1062.659,A -85,B 0,C 180,E1 28155.552,E2 28155.552} C_VEL
LIN {X 0,Y 165.732,Z 1063.807,A -85,B 0,C 180,E1 28161.224,E2 28161.224} C_VEL
LIN {X 0,Y 161.692,Z 1064.035,A -85,B 0,C 180,E1 28167.215,E2 28167.215} C_VEL
LIN {X 0,Y 162.281,Z 1063.211,A -85,B 0,C 180,E1 28175.361,E2 28175.361} C_VEL
LIN {X 0,Y 167.615,Z 1057.418,A -85,B 0,C 180,E1 28191.203,E2 28191.203} C_VEL
LIN {X 0,Y 181.685,Z 1045.916,A -85,B 0,C 180,E1 28205.725,E2 28205.725} C_VEL
LIN {X 0,Y 205.509,Z 1026.916,A -85,B 0,C 180,E1 28218.412,E2 28218.412} C_VEL
LIN {X 0,Y 233.653,Z 1002.441,A -85,B 0,C 180,E1 28227.476,E2 28227.476} C_VEL
LIN {X 0,Y 263.253,Z 972.352,A -85,B 0,C 180,E1 28234.04,E2 28234.04} C_VEL
LIN {X 0,Y 292.497,Z 936.319,A -85,B 0,C 180,E1 28238.842,E2 28238.842} C_VEL
LIN {X 0,Y 297.489,Z 929.115,A -85,B 0,C 180,E1 28239.577,E2 28239.577} C_VEL
LIN {X 0,Y 300.004,Z 915.793,A -85,B 0,C 180,E1 28245.366,E2 28245.366} C_VEL
LIN {X 0,Y 301.348,Z 906.584,A -85,B 0,C 180,E1 28251.499,E2 28251.499} C_VEL
LIN {X 0,Y 302.512,Z 902.126,A -85,B 0,C 180,E1 28257.123,E2 28257.123} C_VEL
LIN {X 0,Y 302.857,Z 901.859,A -85,B 0,C 180,E1 28259.995,E2 28259.995} C_VEL
LIN {X 0,Y 302.425,Z 906.317,A -85,B 0,C 180,E1 28265.746,E2 28265.746} C_VEL
LIN {X 0,Y 301.955,Z 915.259,A -85,B 0,C 180,E1 28271.575,E2 28271.575} C_VEL
LIN {X 0,Y 300.734,Z 927.088,A -85,B 0,C 180,E1 28276.777,E2 28276.777} C_VEL
LIN {X 0,Y 299.026,Z 930.328,A -85,B 0,C 180,E1 28277.336,E2 28277.336} C_VEL
LIN {X 0,Y 271.741,Z 966.389,A -85,B 0,C 180,E1 28281.323,E2 28281.323} C_VEL
LIN {X 0,Y 241.071,Z 999.753,A -85,B 0,C 180,E1 28287.384,E2 28287.384} C_VEL
LIN {X 0,Y 212.673,Z 1026.06,A -85,B 0,C 180,E1 28295.409,E2 28295.409} C_VEL
LIN {X 0,Y 187.651,Z 1047.092,A -85,B 0,C 180,E1 28306.606,E2 28306.606} C_VEL
LIN {X 0,Y 170.359,Z 1061.745,A -85,B 0,C 180,E1 28320.706,E2 28320.706} C_VEL
LIN {X 0,Y 163.406,Z 1069.264,A -85,B 0,C 180,E1 28333.844,E2 28333.844} C_VEL
LIN {X 0,Y 161.735,Z 1072.209,A -85,B 0,C 180,E1 28344.621,E2 28344.621} C_VEL
LIN {X 0,Y 162.134,Z 1072.73,A -85,B 0,C 180,E1 28349.998,E2 28349.998} C_VEL
LIN {X 0,Y 162.18,Z 1071.811,A -85,B 0,C 180,E1 28360.768,E2 28360.768} C_VEL
LIN {X 0,Y 167.629,Z 1066.547,A -85,B 0,C 180,E1 28375.332,E2 28375.332} C_VEL
LIN {X 0,Y 184.319,Z 1053.746,A -85,B 0,C 180,E1 28391.124,E2 28391.124} C_VEL
LIN {X 0,Y 208.908,Z 1035.221,A -85,B 0,C 180,E1 28402.93,E2 28402.93} C_VEL
LIN {X 0,Y 238.183,Z 1010.939,A -85,B 0,C 180,E1 28411.566,E2 28411.566} C_VEL
LIN {X 0,Y 266.788,Z 983.435,A -85,B 0,C 180,E1 28417.368,E2 28417.368} C_VEL
LIN {X 0,Y 294.755,Z 951.429,A -85,B 0,C 180,E1 28421.644,E2 28421.644} C_VEL
LIN {X 0,Y 306.973,Z 935.184,A -85,B 0,C 180,E1 28423.214,E2 28423.214} C_VEL
LIN {X 0,Y 308.454,Z 924.361,A -85,B 0,C 180,E1 28428.672,E2 28428.672} C_VEL
LIN {X 0,Y 309.111,Z 917.344,A -85,B 0,C 180,E1 28434.378,E2 28434.378} C_VEL
LIN {X 0,Y 309.46,Z 914.796,A -85,B 0,C 180,E1 28440.005,E2 28440.005} C_VEL
LIN {X 0,Y 307.662,Z 920.257,A -85,B 0,C 180,E1 28447.119,E2 28447.119} C_VEL
LIN {X 0,Y 306.008,Z 928.214,A -85,B 0,C 180,E1 28452.319,E2 28452.319} C_VEL
LIN {X 0,Y 303.542,Z 936.969,A -85,B 0,C 180,E1 28456.088,E2 28456.088} C_VEL
LIN {X 0,Y 273.205,Z 973.057,A -85,B 0,C 180,E1 28460.589,E2 28460.589} C_VEL
LIN {X 0,Y 241.577,Z 1003.701,A -85,B 0,C 180,E1 28466.912,E2 28466.912} C_VEL
LIN {X 0,Y 211.811,Z 1027.955,A -85,B 0,C 180,E1 28475.506,E2 28475.506} C_VEL
LIN {X 0,Y 185.785,Z 1046.722,A -85,B 0,C 180,E1 28487.743,E2 28487.743} C_VEL
LIN {X 0,Y 170.601,Z 1057.253,A -85,B 0,C 180,E1 28500.757,E2 28500.757} C_VEL
LIN {X 0,Y 162.963,Z 1062.935,A -85,B 0,C 180,E1 28515.261,E2 28515.261} C_VEL
LIN {X 0,Y 161.692,Z 1064.035,A -85,B 0,C 180,E1 28527.215,E2 28527.215} C_VEL
LIN {X 0,Y 159.423,Z 1063.909,A -85,B 0,C 180,E1 28531.818,E2 28531.818} C_VEL
LIN {X 0,Y 154.924,Z 1062.471,A -85,B 0,C 180,E1 28539.747,E2 28539.747} C_VEL
LIN {X 0,Y 162.049,Z 1056.14,A -85,B 0,C 180,E1 28554.889,E2 28554.889} C_VEL
LIN {X 0,Y 178.327,Z 1043.806,A -85,B 0,C 180,E1 28569.307,E2 28569.307} C_VEL
LIN {X 0,Y 201.915,Z 1025.838,A -85,B 0,C 180,E1 28580.774,E2 28580.774} C_VEL
LIN {X 0,Y 230.775,Z 1001.479,A -85,B 0,C 180,E1 28589.515,E2 28589.515} C_VEL
LIN {X 0,Y 260.544,Z 971.946,A -85,B 0,C 180,E1 28595.751,E2 28595.751} C_VEL
LIN {X 0,Y 289.724,Z 936.695,A -85,B 0,C 180,E1 28600.307,E2 28600.307} C_VEL
LIN {X 0,Y 292.667,Z 932.224,A -85,B 0,C 180,E1 28600.9,E2 28600.9} C_VEL
LIN {X 0,Y 295.497,Z 919.391,A -85,B 0,C 180,E1 28607.008,E2 28607.008} C_VEL
LIN {X 0,Y 296.986,Z 911.991,A -85,B 0,C 180,E1 28612.666,E2 28612.666} C_VEL
LIN {X 0,Y 298.012,Z 908.743,A -85,B 0,C 180,E1 28617.08,E2 28617.08} C_VEL
LIN {X 0,Y 298.384,Z 908.429,A -85,B 0,C 180,E1 28619.995,E2 28619.995} C_VEL
LIN {X 0,Y 297.854,Z 913.059,A -85,B 0,C 180,E1 28625.835,E2 28625.835} C_VEL
LIN {X 0,Y 296.869,Z 922.193,A -85,B 0,C 180,E1 28631.776,E2 28631.776} C_VEL
LIN {X 0,Y 295.751,Z 930.491,A -85,B 0,C 180,E1 28635.551,E2 28635.551} C_VEL
LIN {X 0,Y 293.658,Z 934.229,A -85,B 0,C 180,E1 28636.227,E2 28636.227} C_VEL
LIN {X 0,Y 267.215,Z 967.917,A -85,B 0,C 180,E1 28639.972,E2 28639.972} C_VEL
LIN {X 0,Y 237.414,Z 999.436,A -85,B 0,C 180,E1 28645.628,E2 28645.628} C_VEL
LIN {X 0,Y 207.681,Z 1026.074,A -85,B 0,C 180,E1 28653.69,E2 28653.69} C_VEL
LIN {X 0,Y 181.783,Z 1046.817,A -85,B 0,C 180,E1 28664.831,E2 28664.831} C_VEL
LIN {X 0,Y 163.319,Z 1061.494,A -85,B 0,C 180,E1 28679.311,E2 28679.311} C_VEL
LIN {X 0,Y 155.718,Z 1069.03,A -85,B 0,C 180,E1 28693.023,E2 28693.023} C_VEL
LIN {X 0,Y 153.826,Z 1071.988,A -85,B 0,C 180,E1 28704.344,E2 28704.344} C_VEL
LIN {X 0,Y 154.217,Z 1072.516,A -85,B 0,C 180,E1 28709.997,E2 28709.997} C_VEL
LIN {X 0,Y 154.351,Z 1071.607,A -85,B 0,C 180,E1 28721.321,E2 28721.321} C_VEL
LIN {X 0,Y 160.063,Z 1066.546,A -85,B 0,C 180,E1 28736.153,E2 28736.153} C_VEL
LIN {X 0,Y 176.459,Z 1054.742,A -85,B 0,C 180,E1 28751.722,E2 28751.722} C_VEL
LIN {X 0,Y 201.954,Z 1036.599,A -85,B 0,C 180,E1 28764.002,E2 28764.002} C_VEL
LIN {X 0,Y 230.571,Z 1014.072,A -85,B 0,C 180,E1 28772.412,E2 28772.412} C_VEL
LIN {X 0,Y 260.655,Z 986.554,A -85,B 0,C 180,E1 28778.463,E2 28778.463} C_VEL
LIN {X 0,Y 291.643,Z 952.24,A -85,B 0,C 180,E1 28783.05,E2 28783.05} C_VEL
LIN {X 0,Y 301.941,Z 939.063,A -85,B 0,C 180,E1 28784.299,E2 28784.299} C_VEL
LIN {X 0,Y 303.618,Z 928.829,A -85,B 0,C 180,E1 28789.943,E2 28789.943} C_VEL
LIN {X 0,Y 304.334,Z 923.416,A -85,B 0,C 180,E1 28794.781,E2 28794.781} C_VEL
LIN {X 0,Y 304.683,Z 921.177,A -85,B 0,C 180,E1 28800.005,E2 28800.005} C_VEL
LIN {X 0,Y 302.661,Z 926.78,A -85,B 0,C 180,E1 28807.238,E2 28807.238} C_VEL
LIN {X 0,Y 300.221,Z 936.227,A -85,B 0,C 180,E1 28813.134,E2 28813.134} C_VEL
LIN {X 0,Y 299.247,Z 939.429,A -85,B 0,C 180,E1 28814.672,E2 28814.672} C_VEL
LIN {X 0,Y 281.138,Z 961.599,A -85,B 0,C 180,E1 28817.352,E2 28817.352} C_VEL
LIN {X 0,Y 250.29,Z 992.957,A -85,B 0,C 180,E1 28822.587,E2 28822.587} C_VEL
LIN {X 0,Y 217.458,Z 1020.446,A -85,B 0,C 180,E1 28830.42,E2 28830.42} C_VEL
LIN {X 0,Y 189.736,Z 1040.273,A -85,B 0,C 180,E1 28840.649,E2 28840.649} C_VEL
LIN {X 0,Y 167.522,Z 1054.924,A -85,B 0,C 180,E1 28855.244,E2 28855.244} C_VEL
LIN {X 0,Y 158.146,Z 1061.201,A -85,B 0,C 180,E1 28867.465,E2 28867.465} C_VEL
LIN {X 0,Y 154.194,Z 1064.02,A -85,B 0,C 180,E1 28879.406,E2 28879.406} C_VEL
LIN {X 0,Y 154.176,Z 1064.161,A -85,B 0,C 180,E1 28890.003,E2 28890.003} C_VEL
LIN {X 0,Y 154.924,Z 1062.471,A -85,B 0,C 180,E1 28899.747,E2 28899.747} C_VEL
LIN {X 0,Y 153.017,Z 1060.746,A -85,B 0,C 180,E1 28906.196,E2 28906.196} C_VEL
LIN {X 0,Y 152.427,Z 1058.204,A -85,B 0,C 180,E1 28912.752,E2 28912.752} C_VEL
